LIN {X 0,Y 303.808,Z 469.093,A -85,B 0,C 180,E1 -15922.691,E2 -15922.691} C_VEL
LIN {X 0,Y 303.618,Z 471.715,A -85,B 0,C 180,E1 -15924.688,E2 -15924.688} C_VEL
LIN {X 0,Y 303.612,Z 472.958,A -85,B 0,C 180,E1 -15926.018,E2 -15926.018} C_VEL
LIN {X 0,Y 303.631,Z 473.753,A -85,B 0,C 180,E1 -15927.347,E2 -15927.347} C_VEL
LIN {X 0,Y 303.609,Z 474.149,A -85,B 0,C 180,E1 -15928.674,E2 -15928.674} C_VEL
LIN {X 0,Y 303.653,Z 474.153,A -85,B 0,C 180,E1 -15930,E2 -15930} C_VEL
LIN {X 0,Y 303.62,Z 473.754,A -85,B 0,C 180,E1 -15931.326,E2 -15931.326} C_VEL
LIN {X 0,Y 303.636,Z 472.908,A -85,B 0,C 180,E1 -15932.653,E2 -15932.653} C_VEL
LIN {X 0,Y 303.645,Z 471.649,A -85,B 0,C 180,E1 -15933.982,E2 -15933.982} C_VEL
LIN {X 0,Y 303.681,Z 469.543,A -85,B 0,C 180,E1 -15935.611,E2 -15935.611} C_VEL
LIN {X 0,Y 303.944,Z 465.201,A -85,B 0,C 180,E1 -15937.975,E2 -15937.975} C_VEL
LIN {X 0,Y 304.361,Z 460.303,A -85,B 0,C 180,E1 -15939.973,E2 -15939.973} C_VEL
LIN {X 0,Y 304.994,Z 454.106,A -85,B 0,C 180,E1 -15941.969,E2 -15941.969} C_VEL
LIN {X 0,Y 306.125,Z 446.4,A -85,B 0,C 180,E1 -15943.949,E2 -15943.949} C_VEL
LIN {X 0,Y 307.197,Z 438.485,A -85,B 0,C 180,E1 -15945.593,E2 -15945.593} C_VEL
LIN {X 0,Y 308.389,Z 428.8,A -85,B 0,C 180,E1 -15947.233,E2 -15947.233} C_VEL
LIN {X 0,Y 309.728,Z 418.066,A -85,B 0,C 180,E1 -15948.693,E2 -15948.693} C_VEL
LIN {X 0,Y 310.965,Z 407.709,A -85,B 0,C 180,E1 -15949.816,E2 -15949.816} C_VEL
LIN {X 0,Y 312.28,Z 395.367,A -85,B 0,C 180,E1 -15950.846,E2 -15950.846} C_VEL
LIN {X 0,Y 313.335,Z 382.457,A -85,B 0,C 180,E1 -15951.634,E2 -15951.634} C_VEL
LIN {X 0,Y 314.078,Z 370.101,A -85,B 0,C 180,E1 -15952.142,E2 -15952.142} C_VEL
LIN {X 0,Y 315.753,Z 303.823,A -85,B 0,C 180,E1 -15953.743,E2 -15953.743} C_VEL
LIN {X 0,Y 309.938,Z 264.176,A -85,B 0,C 180,E1 -15955.182,E2 -15955.182} C_VEL
LIN {X 0,Y 309.571,Z 261.875,A -85,B 0,C 180,E1 -15955.29,E2 -15955.29} C_VEL
LIN {X 0,Y 309.852,Z 258.307,A -85,B 0,C 180,E1 -15956.25,E2 -15956.25} C_VEL
LIN {X 0,Y 307.948,Z 247.956,A -85,B 0,C 180,E1 -15959.276,E2 -15959.276} C_VEL
LIN {X 0,Y 305.49,Z 236.432,A -85,B 0,C 180,E1 -15962.824,E2 -15962.824} C_VEL
LIN {X 0,Y 305.461,Z 236.433,A -85,B 0,C 180,E1 -15966.74,E2 -15966.74} C_VEL
LIN {X 0,Y 305.404,Z 236.442,A -85,B 0,C 180,E1 -15970.581,E2 -15970.581} C_VEL
LIN {X 0,Y 305.395,Z 236.443,A -85,B 0,C 180,E1 -15974.481,E2 -15974.481} C_VEL
LIN {X 0,Y 305.398,Z 236.443,A -85,B 0,C 180,E1 -15978.129,E2 -15978.129} C_VEL
LIN {X 0,Y 305.438,Z 236.44,A -85,B 0,C 180,E1 -15981.585,E2 -15981.585} C_VEL
LIN {X 0,Y 305.469,Z 236.432,A -85,B 0,C 180,E1 -15984.881,E2 -15984.881} C_VEL
LIN {X 0,Y 305.446,Z 236.435,A -85,B 0,C 180,E1 -15988.355,E2 -15988.355} C_VEL
LIN {X 0,Y 305.456,Z 236.435,A -85,B 0,C 180,E1 -15991.101,E2 -15991.101} C_VEL
LIN {X 0,Y 305.484,Z 236.431,A -85,B 0,C 180,E1 -15994.073,E2 -15994.073} C_VEL
LIN {X 0,Y 305.462,Z 236.431,A -85,B 0,C 180,E1 -15998.393,E2 -15998.393} C_VEL
LIN {X 0,Y 305.521,Z 236.418,A -85,B 0,C 180,E1 -16002.593,E2 -16002.593} C_VEL
LIN {X 0,Y 305.626,Z 236.412,A -85,B 0,C 180,E1 -16005.341,E2 -16005.341} C_VEL
LIN {X 0,Y 305.618,Z 236.417,A -85,B 0,C 180,E1 -16009.392,E2 -16009.392} C_VEL
LIN {X 0,Y 305.734,Z 236.397,A -85,B 0,C 180,E1 -16012.065,E2 -16012.065} C_VEL
LIN {X 0,Y 305.646,Z 236.404,A -85,B 0,C 180,E1 -16014.716,E2 -16014.716} C_VEL
LIN {X 0,Y 305.933,Z 236.367,A -85,B 0,C 180,E1 -16018.676,E2 -16018.676} C_VEL
LIN {X 0,Y 305.925,Z 236.375,A -85,B 0,C 180,E1 -16021.309,E2 -16021.309} C_VEL
LIN {X 0,Y 305.645,Z 236.413,A -85,B 0,C 180,E1 -16025.269,E2 -16025.269} C_VEL
LIN {X 0,Y 305.73,Z 236.399,A -85,B 0,C 180,E1 -16027.92,E2 -16027.92} C_VEL
LIN {X 0,Y 305.579,Z 236.419,A -85,B 0,C 180,E1 -16031.938,E2 -16031.938} C_VEL
LIN {X 0,Y 305.59,Z 236.418,A -85,B 0,C 180,E1 -16035.006,E2 -16035.006} C_VEL
LIN {X 0,Y 305.539,Z 236.425,A -85,B 0,C 180,E1 -16039.428,E2 -16039.428} C_VEL
LIN {X 0,Y 305.462,Z 236.434,A -85,B 0,C 180,E1 -16043.032,E2 -16043.032} C_VEL
LIN {X 0,Y 305.473,Z 236.429,A -85,B 0,C 180,E1 -16046.201,E2 -16046.201} C_VEL
LIN {X 0,Y 305.446,Z 236.432,A -85,B 0,C 180,E1 -16049.035,E2 -16049.035} C_VEL
LIN {X 0,Y 305.431,Z 236.435,A -85,B 0,C 180,E1 -16053.51,E2 -16053.51} C_VEL
LIN {X 0,Y 305.42,Z 236.437,A -85,B 0,C 180,E1 -16056.735,E2 -16056.735} C_VEL
LIN {X 0,Y 305.416,Z 236.439,A -85,B 0,C 180,E1 -16060.593,E2 -16060.593} C_VEL
LIN {X 0,Y 305.376,Z 236.442,A -85,B 0,C 180,E1 -16064.486,E2 -16064.486} C_VEL
LIN {X 0,Y 305.397,Z 236.44,A -85,B 0,C 180,E1 -16068.137,E2 -16068.137} C_VEL
LIN {X 0,Y 305.429,Z 236.439,A -85,B 0,C 180,E1 -16071.592,E2 -16071.592} C_VEL
LIN {X 0,Y 305.413,Z 236.441,A -85,B 0,C 180,E1 -16074.881,E2 -16074.881} C_VEL
LIN {X 0,Y 305.401,Z 236.44,A -85,B 0,C 180,E1 -16078.351,E2 -16078.351} C_VEL
LIN {X 0,Y 305.469,Z 236.437,A -85,B 0,C 180,E1 -16081.109,E2 -16081.109} C_VEL
LIN {X 0,Y 305.521,Z 236.426,A -85,B 0,C 180,E1 -16084.084,E2 -16084.084} C_VEL
LIN {X 0,Y 305.494,Z 236.429,A -85,B 0,C 180,E1 -16088.403,E2 -16088.403} C_VEL
LIN {X 0,Y 305.538,Z 236.428,A -85,B 0,C 180,E1 -16091.215,E2 -16091.215} C_VEL
LIN {X 0,Y 305.592,Z 236.419,A -85,B 0,C 180,E1 -16095.347,E2 -16095.347} C_VEL
LIN {X 0,Y 305.583,Z 236.42,A -85,B 0,C 180,E1 -16099.398,E2 -16099.398} C_VEL
LIN {X 0,Y 305.758,Z 236.395,A -85,B 0,C 180,E1 -16102.073,E2 -16102.073} C_VEL
LIN {X 0,Y 305.639,Z 236.413,A -85,B 0,C 180,E1 -16104.723,E2 -16104.723} C_VEL
LIN {X 0,Y 305.905,Z 236.38,A -85,B 0,C 180,E1 -16108.683,E2 -16108.683} C_VEL
LIN {X 0,Y 305.905,Z 236.38,A -85,B 0,C 180,E1 -16111.316,E2 -16111.316} C_VEL
LIN {X 0,Y 305.767,Z 236.478,A -85,B 0,C 180,E1 -16116.143,E2 -16116.143} C_VEL
LIN {X 0,Y 306.706,Z 241.054,A -85,B 0,C 180,E1 -16117.592,E2 -16117.592} C_VEL
LIN {X 0,Y 315.156,Z 264.98,A -85,B 0,C 180,E1 -16118.847,E2 -16118.847} C_VEL
LIN {X 0,Y 316.427,Z 271.959,A -85,B 0,C 180,E1 -16119.115,E2 -16119.115} C_VEL
LIN {X 0,Y 314.322,Z 348.83,A -85,B 0,C 180,E1 -16120.97,E2 -16120.97} C_VEL
LIN {X 0,Y 313.559,Z 362.432,A -85,B 0,C 180,E1 -16121.565,E2 -16121.565} C_VEL
LIN {X 0,Y 312.712,Z 375.269,A -85,B 0,C 180,E1 -16122.41,E2 -16122.41} C_VEL
LIN {X 0,Y 311.564,Z 387.718,A -85,B 0,C 180,E1 -16123.523,E2 -16123.523} C_VEL
LIN {X 0,Y 310.355,Z 398.515,A -85,B 0,C 180,E1 -16124.759,E2 -16124.759} C_VEL
LIN {X 0,Y 309.13,Z 408.276,A -85,B 0,C 180,E1 -16126.148,E2 -16126.148} C_VEL
LIN {X 0,Y 307.919,Z 416.664,A -85,B 0,C 180,E1 -16127.602,E2 -16127.602} C_VEL
LIN {X 0,Y 306.806,Z 425.084,A -85,B 0,C 180,E1 -16129.399,E2 -16129.399} C_VEL
LIN {X 0,Y 305.666,Z 433.288,A -85,B 0,C 180,E1 -16131.584,E2 -16131.584} C_VEL
LIN {X 0,Y 304.82,Z 439.711,A -85,B 0,C 180,E1 -16133.795,E2 -16133.795} C_VEL
LIN {X 0,Y 304.268,Z 444.645,A -85,B 0,C 180,E1 -16136.03,E2 -16136.03} C_VEL
LIN {X 0,Y 304.04,Z 447.221,A -85,B 0,C 180,E1 -16137.535,E2 -16137.535} C_VEL
LIN {X 0,Y 303.695,Z 449.214,A -85,B 0,C 180,E1 -16139.075,E2 -16139.075} C_VEL
LIN {X 0,Y 303.446,Z 450.963,A -85,B 0,C 180,E1 -16141.045,E2 -16141.045} C_VEL
LIN {X 0,Y 303.388,Z 451.891,A -85,B 0,C 180,E1 -16143.513,E2 -16143.513} C_VEL
LIN {X 0,Y 303.557,Z 451.493,A -85,B 0,C 180,E1 -16145.89,E2 -16145.89} C_VEL
LIN {X 0,Y 303.919,Z 449.867,A -85,B 0,C 180,E1 -16148.181,E2 -16148.181} C_VEL
LIN {X 0,Y 304.479,Z 447.101,A -85,B 0,C 180,E1 -16150.401,E2 -16150.401} C_VEL
LIN {X 0,Y 305.174,Z 443.252,A -85,B 0,C 180,E1 -16152.543,E2 -16152.543} C_VEL
LIN {X 0,Y 306.16,Z 438.196,A -85,B 0,C 180,E1 -16154.648,E2 -16154.648} C_VEL
LIN {X 0,Y 307.427,Z 431.82,A -85,B 0,C 180,E1 -16156.713,E2 -16156.713} C_VEL
LIN {X 0,Y 308.973,Z 423.866,A -85,B 0,C 180,E1 -16158.74,E2 -16158.74} C_VEL
LIN {X 0,Y 310.631,Z 414.677,A -85,B 0,C 180,E1 -16160.599,E2 -16160.599} C_VEL
LIN {X 0,Y 312.313,Z 405.038,A -85,B 0,C 180,E1 -16162.166,E2 -16162.166} C_VEL
LIN {X 0,Y 313.851,Z 394.716,A -85,B 0,C 180,E1 -16163.516,E2 -16163.516} C_VEL
LIN {X 0,Y 315.441,Z 382.749,A -85,B 0,C 180,E1 -16164.74,E2 -16164.74} C_VEL
LIN {X 0,Y 316.716,Z 370.283,A -85,B 0,C 180,E1 -16165.717,E2 -16165.717} C_VEL
LIN {X 0,Y 317.728,Z 357.146,A -85,B 0,C 180,E1 -16166.439,E2 -16166.439} C_VEL
LIN {X 0,Y 318.347,Z 344.513,A -85,B 0,C 180,E1 -16166.887,E2 -16166.887} C_VEL
LIN {X 0,Y 318.017,Z 338.724,A -85,B 0,C 180,E1 -16167.093,E2 -16167.093} C_VEL
LIN {X 0,Y 313.501,Z 320.095,A -85,B 0,C 180,E1 -16168.037,E2 -16168.037} C_VEL
LIN {X 0,Y 313.101,Z 314.293,A -85,B 0,C 180,E1 -16168.235,E2 -16168.235} C_VEL
LIN {X 0,Y 314.444,Z 274.419,A -85,B 0,C 180,E1 -16169.216,E2 -16169.216} C_VEL
LIN {X 0,Y 309.017,Z 261.151,A -85,B 0,C 180,E1 -16170.202,E2 -16170.202} C_VEL
LIN {X 0,Y 302.527,Z 247.643,A -85,B 0,C 180,E1 -16171.381,E2 -16171.381} C_VEL
LIN {X 0,Y 299.66,Z 242.008,A -85,B 0,C 180,E1 -16171.942,E2 -16171.942} C_VEL
LIN {X 0,Y 298.473,Z 237.305,A -85,B 0,C 180,E1 -16173.695,E2 -16173.695} C_VEL
LIN {X 0,Y 298.405,Z 237.314,A -85,B 0,C 180,E1 -16177.872,E2 -16177.872} C_VEL
LIN {X 0,Y 298.516,Z 237.302,A -85,B 0,C 180,E1 -16180.765,E2 -16180.765} C_VEL
LIN {X 0,Y 298.574,Z 237.292,A -85,B 0,C 180,E1 -16185.003,E2 -16185.003} C_VEL
LIN {X 0,Y 298.576,Z 237.292,A -85,B 0,C 180,E1 -16189.154,E2 -16189.154} C_VEL
LIN {X 0,Y 298.702,Z 237.272,A -85,B 0,C 180,E1 -16191.893,E2 -16191.893} C_VEL
LIN {X 0,Y 298.633,Z 237.281,A -85,B 0,C 180,E1 -16194.606,E2 -16194.606} C_VEL
LIN {X 0,Y 298.91,Z 237.245,A -85,B 0,C 180,E1 -16198.66,E2 -16198.66} C_VEL
LIN {X 0,Y 298.907,Z 237.245,A -85,B 0,C 180,E1 -16201.355,E2 -16201.355} C_VEL
LIN {X 0,Y 298.748,Z 237.264,A -85,B 0,C 180,E1 -16206.762,E2 -16206.762} C_VEL
LIN {X 0,Y 298.623,Z 237.279,A -85,B 0,C 180,E1 -16209.489,E2 -16209.489} C_VEL
LIN {X 0,Y 298.543,Z 237.291,A -85,B 0,C 180,E1 -16213.623,E2 -16213.623} C_VEL
LIN {X 0,Y 298.485,Z 237.306,A -85,B 0,C 180,E1 -16216.419,E2 -16216.419} C_VEL
LIN {X 0,Y 298.443,Z 237.306,A -85,B 0,C 180,E1 -16219.622,E2 -16219.622} C_VEL
LIN {X 0,Y 298.389,Z 237.312,A -85,B 0,C 180,E1 -16223.61,E2 -16223.61} C_VEL
LIN {X 0,Y 298.407,Z 237.306,A -85,B 0,C 180,E1 -16226.589,E2 -16226.589} C_VEL
LIN {X 0,Y 298.363,Z 237.313,A -85,B 0,C 180,E1 -16229.654,E2 -16229.654} C_VEL
LIN {X 0,Y 298.4,Z 237.31,A -85,B 0,C 180,E1 -16232.806,E2 -16232.806} C_VEL
LIN {X 0,Y 298.412,Z 237.312,A -85,B 0,C 180,E1 -16236.078,E2 -16236.078} C_VEL
LIN {X 0,Y 298.355,Z 237.317,A -85,B 0,C 180,E1 -16239.502,E2 -16239.502} C_VEL
LIN {X 0,Y 298.353,Z 237.324,A -85,B 0,C 180,E1 -16243.096,E2 -16243.096} C_VEL
LIN {X 0,Y 298.354,Z 237.323,A -85,B 0,C 180,E1 -16246.913,E2 -16246.913} C_VEL
LIN {X 0,Y 298.376,Z 237.318,A -85,B 0,C 180,E1 -16251.021,E2 -16251.021} C_VEL
LIN {X 0,Y 298.522,Z 237.477,A -85,B 0,C 180,E1 -16254.14,E2 -16254.14} C_VEL
LIN {X 0,Y 301.257,Z 248.367,A -85,B 0,C 180,E1 -16257.946,E2 -16257.946} C_VEL
LIN {X 0,Y 303.213,Z 257.381,A -85,B 0,C 180,E1 -16260.874,E2 -16260.874} C_VEL
LIN {X 0,Y 303.756,Z 260.098,A -85,B 0,C 180,E1 -16261.647,E2 -16261.647} C_VEL
LIN {X 0,Y 307.237,Z 268.773,A -85,B 0,C 180,E1 -16262.317,E2 -16262.317} C_VEL
LIN {X 0,Y 311.274,Z 289.894,A -85,B 0,C 180,E1 -16263.383,E2 -16263.383} C_VEL
LIN {X 0,Y 313.497,Z 306.34,A -85,B 0,C 180,E1 -16264.084,E2 -16264.084} C_VEL
LIN {X 0,Y 311.413,Z 369.696,A -85,B 0,C 180,E1 -16265.674,E2 -16265.674} C_VEL
LIN {X 0,Y 310.328,Z 383.207,A -85,B 0,C 180,E1 -16266.254,E2 -16266.254} C_VEL
LIN {X 0,Y 308.956,Z 395.991,A -85,B 0,C 180,E1 -16267.074,E2 -16267.074} C_VEL
LIN {X 0,Y 307.42,Z 406.931,A -85,B 0,C 180,E1 -16268.016,E2 -16268.016} C_VEL
LIN {X 0,Y 305.646,Z 418.42,A -85,B 0,C 180,E1 -16269.297,E2 -16269.297} C_VEL
LIN {X 0,Y 303.855,Z 428.82,A -85,B 0,C 180,E1 -16270.756,E2 -16270.756} C_VEL
LIN {X 0,Y 302.135,Z 438.215,A -85,B 0,C 180,E1 -16272.399,E2 -16272.399} C_VEL
LIN {X 0,Y 300.481,Z 447.324,A -85,B 0,C 180,E1 -16274.397,E2 -16274.397} C_VEL
LIN {X 0,Y 299.002,Z 454.708,A -85,B 0,C 180,E1 -16276.406,E2 -16276.406} C_VEL
LIN {X 0,Y 297.913,Z 460.651,A -85,B 0,C 180,E1 -16278.433,E2 -16278.433} C_VEL
LIN {X 0,Y 297.22,Z 465.351,A -85,B 0,C 180,E1 -16280.473,E2 -16280.473} C_VEL
LIN {X 0,Y 296.738,Z 468.945,A -85,B 0,C 180,E1 -16282.515,E2 -16282.515} C_VEL
LIN {X 0,Y 296.533,Z 471.531,A -85,B 0,C 180,E1 -16284.56,E2 -16284.56} C_VEL
LIN {X 0,Y 296.511,Z 472.744,A -85,B 0,C 180,E1 -16285.923,E2 -16285.923} C_VEL
LIN {X 0,Y 296.555,Z 473.516,A -85,B 0,C 180,E1 -16287.283,E2 -16287.283} C_VEL
LIN {X 0,Y 296.527,Z 473.893,A -85,B 0,C 180,E1 -16288.642,E2 -16288.642} C_VEL
LIN {X 0,Y 296.567,Z 473.88,A -85,B 0,C 180,E1 -16290,E2 -16290} C_VEL
LIN {X 0,Y 296.538,Z 473.454,A -85,B 0,C 180,E1 -16291.358,E2 -16291.358} C_VEL
LIN {X 0,Y 296.562,Z 472.584,A -85,B 0,C 180,E1 -16292.717,E2 -16292.717} C_VEL
LIN {X 0,Y 296.544,Z 471.305,A -85,B 0,C 180,E1 -16294.077,E2 -16294.077} C_VEL
LIN {X 0,Y 296.609,Z 469.4,A -85,B 0,C 180,E1 -16295.592,E2 -16295.592} C_VEL
LIN {X 0,Y 296.795,Z 466.181,A -85,B 0,C 180,E1 -16297.483,E2 -16297.483} C_VEL
LIN {X 0,Y 297.152,Z 461.638,A -85,B 0,C 180,E1 -16299.53,E2 -16299.53} C_VEL
LIN {X 0,Y 297.736,Z 455.847,A -85,B 0,C 180,E1 -16301.574,E2 -16301.574} C_VEL
LIN {X 0,Y 298.792,Z 448.573,A -85,B 0,C 180,E1 -16303.604,E2 -16303.604} C_VEL
LIN {X 0,Y 300.074,Z 439.516,A -85,B 0,C 180,E1 -16305.625,E2 -16305.625} C_VEL
LIN {X 0,Y 301.234,Z 430.332,A -85,B 0,C 180,E1 -16307.278,E2 -16307.278} C_VEL
LIN {X 0,Y 302.669,Z 419.78,A -85,B 0,C 180,E1 -16308.794,E2 -16308.794} C_VEL
LIN {X 0,Y 304.075,Z 408.261,A -85,B 0,C 180,E1 -16310.108,E2 -16310.108} C_VEL
LIN {X 0,Y 305.407,Z 396.25,A -85,B 0,C 180,E1 -16311.161,E2 -16311.161} C_VEL
LIN {X 0,Y 306.541,Z 382.972,A -85,B 0,C 180,E1 -16312.006,E2 -16312.006} C_VEL
LIN {X 0,Y 307.353,Z 369.883,A -85,B 0,C 180,E1 -16312.564,E2 -16312.564} C_VEL
LIN {X 0,Y 309.013,Z 304.065,A -85,B 0,C 180,E1 -16314.194,E2 -16314.194} C_VEL
LIN {X 0,Y 302.799,Z 261.719,A -85,B 0,C 180,E1 -16315.784,E2 -16315.784} C_VEL
LIN {X 0,Y 302.622,Z 257.699,A -85,B 0,C 180,E1 -16316.927,E2 -16316.927} C_VEL
LIN {X 0,Y 300.354,Z 246.078,A -85,B 0,C 180,E1 -16320.447,E2 -16320.447} C_VEL
LIN {X 0,Y 298.446,Z 237.311,A -85,B 0,C 180,E1 -16323.296,E2 -16323.296} C_VEL
LIN {X 0,Y 298.436,Z 237.308,A -85,B 0,C 180,E1 -16326.797,E2 -16326.797} C_VEL
LIN {X 0,Y 298.345,Z 237.322,A -85,B 0,C 180,E1 -16331.071,E2 -16331.071} C_VEL
LIN {X 0,Y 298.339,Z 237.322,A -85,B 0,C 180,E1 -16335.025,E2 -16335.025} C_VEL
LIN {X 0,Y 298.346,Z 237.319,A -85,B 0,C 180,E1 -16338.92,E2 -16338.92} C_VEL
LIN {X 0,Y 298.434,Z 237.31,A -85,B 0,C 180,E1 -16343.194,E2 -16343.194} C_VEL
LIN {X 0,Y 298.417,Z 237.315,A -85,B 0,C 180,E1 -16345.575,E2 -16345.575} C_VEL
LIN {X 0,Y 298.375,Z 237.315,A -85,B 0,C 180,E1 -16348.782,E2 -16348.782} C_VEL
LIN {X 0,Y 298.4,Z 237.315,A -85,B 0,C 180,E1 -16351.891,E2 -16351.891} C_VEL
LIN {X 0,Y 298.427,Z 237.309,A -85,B 0,C 180,E1 -16354.912,E2 -16354.912} C_VEL
LIN {X 0,Y 298.396,Z 237.314,A -85,B 0,C 180,E1 -16357.855,E2 -16357.855} C_VEL
LIN {X 0,Y 298.456,Z 237.3,A -85,B 0,C 180,E1 -16360.744,E2 -16360.744} C_VEL
LIN {X 0,Y 298.588,Z 237.286,A -85,B 0,C 180,E1 -16364.988,E2 -16364.988} C_VEL
LIN {X 0,Y 298.578,Z 237.292,A -85,B 0,C 180,E1 -16369.139,E2 -16369.139} C_VEL
LIN {X 0,Y 298.68,Z 237.277,A -85,B 0,C 180,E1 -16371.877,E2 -16371.877} C_VEL
LIN {X 0,Y 298.617,Z 237.278,A -85,B 0,C 180,E1 -16374.591,E2 -16374.591} C_VEL
LIN {X 0,Y 298.899,Z 237.242,A -85,B 0,C 180,E1 -16378.645,E2 -16378.645} C_VEL
LIN {X 0,Y 298.893,Z 237.251,A -85,B 0,C 180,E1 -16381.34,E2 -16381.34} C_VEL
LIN {X 0,Y 298.718,Z 237.273,A -85,B 0,C 180,E1 -16386.748,E2 -16386.748} C_VEL
LIN {X 0,Y 298.61,Z 237.287,A -85,B 0,C 180,E1 -16389.474,E2 -16389.474} C_VEL
LIN {X 0,Y 298.525,Z 237.3,A -85,B 0,C 180,E1 -16393.608,E2 -16393.608} C_VEL
LIN {X 0,Y 298.466,Z 237.303,A -85,B 0,C 180,E1 -16396.404,E2 -16396.404} C_VEL
LIN {X 0,Y 298.476,Z 237.304,A -85,B 0,C 180,E1 -16399.639,E2 -16399.639} C_VEL
LIN {X 0,Y 298.4,Z 237.315,A -85,B 0,C 180,E1 -16403.593,E2 -16403.593} C_VEL
LIN {X 0,Y 298.427,Z 237.306,A -85,B 0,C 180,E1 -16406.57,E2 -16406.57} C_VEL
LIN {X 0,Y 298.377,Z 237.307,A -85,B 0,C 180,E1 -16409.635,E2 -16409.635} C_VEL
LIN {X 0,Y 298.36,Z 237.307,A -85,B 0,C 180,E1 -16412.793,E2 -16412.793} C_VEL
LIN {X 0,Y 298.394,Z 237.312,A -85,B 0,C 180,E1 -16416.796,E2 -16416.796} C_VEL
LIN {X 0,Y 298.349,Z 237.322,A -85,B 0,C 180,E1 -16421.081,E2 -16421.081} C_VEL
LIN {X 0,Y 298.359,Z 237.32,A -85,B 0,C 180,E1 -16423.097,E2 -16423.097} C_VEL
LIN {X 0,Y 298.361,Z 237.319,A -85,B 0,C 180,E1 -16426.915,E2 -16426.915} C_VEL
LIN {X 0,Y 298.358,Z 237.318,A -85,B 0,C 180,E1 -16431.001,E2 -16431.001} C_VEL
LIN {X 0,Y 298.37,Z 237.317,A -85,B 0,C 180,E1 -16433.924,E2 -16433.924} C_VEL
LIN {X 0,Y 298.345,Z 237.32,A -85,B 0,C 180,E1 -16437.979,E2 -16437.979} C_VEL
LIN {X 0,Y 298.418,Z 237.31,A -85,B 0,C 180,E1 -16441.9,E2 -16441.9} C_VEL
LIN {X 0,Y 298.447,Z 237.311,A -85,B 0,C 180,E1 -16444.921,E2 -16444.921} C_VEL
LIN {X 0,Y 298.423,Z 237.31,A -85,B 0,C 180,E1 -16447.864,E2 -16447.864} C_VEL
LIN {X 0,Y 298.504,Z 237.303,A -85,B 0,C 180,E1 -16450.755,E2 -16450.755} C_VEL
LIN {X 0,Y 298.537,Z 237.301,A -85,B 0,C 180,E1 -16454.992,E2 -16454.992} C_VEL
LIN {X 0,Y 298.538,Z 237.299,A -85,B 0,C 180,E1 -16459.145,E2 -16459.145} C_VEL
LIN {X 0,Y 298.703,Z 237.274,A -85,B 0,C 180,E1 -16461.885,E2 -16461.885} C_VEL
LIN {X 0,Y 298.609,Z 237.288,A -85,B 0,C 180,E1 -16464.598,E2 -16464.598} C_VEL
LIN {X 0,Y 298.871,Z 237.256,A -85,B 0,C 180,E1 -16468.653,E2 -16468.653} C_VEL
LIN {X 0,Y 298.871,Z 237.256,A -85,B 0,C 180,E1 -16471.347,E2 -16471.347} C_VEL
LIN {X 0,Y 298.655,Z 237.315,A -85,B 0,C 180,E1 -16475.74,E2 -16475.74} C_VEL
LIN {X 0,Y 299.529,Z 241.265,A -85,B 0,C 180,E1 -16477.034,E2 -16477.034} C_VEL
LIN {X 0,Y 308.776,Z 267.168,A -85,B 0,C 180,E1 -16478.446,E2 -16478.446} C_VEL
LIN {X 0,Y 309.771,Z 273.543,A -85,B 0,C 180,E1 -16478.685,E2 -16478.685} C_VEL
LIN {X 0,Y 307.638,Z 348.571,A -85,B 0,C 180,E1 -16480.53,E2 -16480.53} C_VEL
LIN {X 0,Y 306.868,Z 361.957,A -85,B 0,C 180,E1 -16481.117,E2 -16481.117} C_VEL
LIN {X 0,Y 306.044,Z 374.352,A -85,B 0,C 180,E1 -16481.927,E2 -16481.927} C_VEL
LIN {X 0,Y 304.91,Z 386.352,A -85,B 0,C 180,E1 -16482.987,E2 -16482.987} C_VEL
LIN {X 0,Y 303.643,Z 397.605,A -85,B 0,C 180,E1 -16484.269,E2 -16484.269} C_VEL
LIN {X 0,Y 302.363,Z 407.51,A -85,B 0,C 180,E1 -16485.676,E2 -16485.676} C_VEL
LIN {X 0,Y 301.03,Z 416.68,A -85,B 0,C 180,E1 -16487.276,E2 -16487.276} C_VEL
LIN {X 0,Y 299.839,Z 425.328,A -85,B 0,C 180,E1 -16489.156,E2 -16489.156} C_VEL
LIN {X 0,Y 298.667,Z 433.533,A -85,B 0,C 180,E1 -16491.39,E2 -16491.39} C_VEL
LIN {X 0,Y 297.779,Z 439.964,A -85,B 0,C 180,E1 -16493.654,E2 -16493.654} C_VEL
LIN {X 0,Y 297.168,Z 445.08,A -85,B 0,C 180,E1 -16496.037,E2 -16496.037} C_VEL
LIN {X 0,Y 296.783,Z 448.544,A -85,B 0,C 180,E1 -16498.268,E2 -16498.268} C_VEL
LIN {X 0,Y 296.49,Z 450.281,A -85,B 0,C 180,E1 -16499.853,E2 -16499.853} C_VEL
LIN {X 0,Y 296.318,Z 451.458,A -85,B 0,C 180,E1 -16501.451,E2 -16501.451} C_VEL
LIN {X 0,Y 296.303,Z 452.196,A -85,B 0,C 180,E1 -16503.903,E2 -16503.903} C_VEL
LIN {X 0,Y 296.51,Z 451.605,A -85,B 0,C 180,E1 -16506.338,E2 -16506.338} C_VEL
LIN {X 0,Y 296.924,Z 449.847,A -85,B 0,C 180,E1 -16508.656,E2 -16508.656} C_VEL
LIN {X 0,Y 297.57,Z 446.95,A -85,B 0,C 180,E1 -16510.922,E2 -16510.922} C_VEL
LIN {X 0,Y 298.356,Z 442.965,A -85,B 0,C 180,E1 -16513.109,E2 -16513.109} C_VEL
LIN {X 0,Y 299.401,Z 437.791,A -85,B 0,C 180,E1 -16515.249,E2 -16515.249} C_VEL
LIN {X 0,Y 300.765,Z 431.26,A -85,B 0,C 180,E1 -16517.354,E2 -16517.354} C_VEL
LIN {X 0,Y 302.419,Z 423.097,A -85,B 0,C 180,E1 -16519.419,E2 -16519.419} C_VEL
LIN {X 0,Y 304.049,Z 414.684,A -85,B 0,C 180,E1 -16521.131,E2 -16521.131} C_VEL
LIN {X 0,Y 305.787,Z 405.006,A -85,B 0,C 180,E1 -16522.728,E2 -16522.728} C_VEL
LIN {X 0,Y 307.441,Z 394.349,A -85,B 0,C 180,E1 -16524.13,E2 -16524.13} C_VEL
LIN {X 0,Y 309.116,Z 382.252,A -85,B 0,C 180,E1 -16525.373,E2 -16525.373} C_VEL
LIN {X 0,Y 310.324,Z 371.025,A -85,B 0,C 180,E1 -16526.262,E2 -16526.262} C_VEL
LIN {X 0,Y 311.385,Z 357.871,A -85,B 0,C 180,E1 -16527.01,E2 -16527.01} C_VEL
LIN {X 0,Y 312.073,Z 344.69,A -85,B 0,C 180,E1 -16527.488,E2 -16527.488} C_VEL
LIN {X 0,Y 313.101,Z 314.293,A -85,B 0,C 180,E1 -16528.235,E2 -16528.235} C_VEL
LIN {X 0,Y 312.723,Z 308.495,A -85,B 0,C 180,E1 -16528.438,E2 -16528.438} C_VEL
LIN {X 0,Y 308.404,Z 289.883,A -85,B 0,C 180,E1 -16529.436,E2 -16529.436} C_VEL
LIN {X 0,Y 308.061,Z 284.086,A -85,B 0,C 180,E1 -16529.642,E2 -16529.642} C_VEL
LIN {X 0,Y 308.218,Z 275.788,A -85,B 0,C 180,E1 -16529.866,E2 -16529.866} C_VEL
LIN {X 0,Y 302.127,Z 261.5,A -85,B 0,C 180,E1 -16531.007,E2 -16531.007} C_VEL
LIN {X 0,Y 296.111,Z 249.265,A -85,B 0,C 180,E1 -16532.153,E2 -16532.153} C_VEL
LIN {X 0,Y 292.491,Z 242.304,A -85,B 0,C 180,E1 -16532.904,E2 -16532.904} C_VEL
LIN {X 0,Y 291.428,Z 238.184,A -85,B 0,C 180,E1 -16534.523,E2 -16534.523} C_VEL
LIN {X 0,Y 291.356,Z 238.194,A -85,B 0,C 180,E1 -16537.307,E2 -16537.307} C_VEL
LIN {X 0,Y 291.436,Z 238.182,A -85,B 0,C 180,E1 -16540.278,E2 -16540.278} C_VEL
LIN {X 0,Y 291.522,Z 238.173,A -85,B 0,C 180,E1 -16544.642,E2 -16544.642} C_VEL
LIN {X 0,Y 291.52,Z 238.169,A -85,B 0,C 180,E1 -16548.889,E2 -16548.889} C_VEL
LIN {X 0,Y 291.652,Z 238.15,A -85,B 0,C 180,E1 -16551.695,E2 -16551.695} C_VEL
LIN {X 0,Y 291.602,Z 238.156,A -85,B 0,C 180,E1 -16554.476,E2 -16554.476} C_VEL
LIN {X 0,Y 291.876,Z 238.12,A -85,B 0,C 180,E1 -16558.628,E2 -16558.628} C_VEL
LIN {X 0,Y 291.873,Z 238.121,A -85,B 0,C 180,E1 -16561.387,E2 -16561.387} C_VEL
LIN {X 0,Y 291.699,Z 238.143,A -85,B 0,C 180,E1 -16566.926,E2 -16566.926} C_VEL
LIN {X 0,Y 291.566,Z 238.157,A -85,B 0,C 180,E1 -16569.721,E2 -16569.721} C_VEL
LIN {X 0,Y 291.514,Z 238.164,A -85,B 0,C 180,E1 -16573.958,E2 -16573.958} C_VEL
LIN {X 0,Y 291.43,Z 238.182,A -85,B 0,C 180,E1 -16576.828,E2 -16576.828} C_VEL
LIN {X 0,Y 291.395,Z 238.184,A -85,B 0,C 180,E1 -16579.849,E2 -16579.849} C_VEL
LIN {X 0,Y 291.334,Z 238.193,A -85,B 0,C 180,E1 -16584.218,E2 -16584.218} C_VEL
LIN {X 0,Y 291.335,Z 238.19,A -85,B 0,C 180,E1 -16587.287,E2 -16587.287} C_VEL
LIN {X 0,Y 291.308,Z 238.191,A -85,B 0,C 180,E1 -16590.447,E2 -16590.447} C_VEL
LIN {X 0,Y 291.352,Z 238.185,A -85,B 0,C 180,E1 -16593.704,E2 -16593.704} C_VEL
LIN {X 0,Y 291.358,Z 238.188,A -85,B 0,C 180,E1 -16597.251,E2 -16597.251} C_VEL
LIN {X 0,Y 291.296,Z 238.201,A -85,B 0,C 180,E1 -16600.656,E2 -16600.656} C_VEL
LIN {X 0,Y 291.288,Z 238.204,A -85,B 0,C 180,E1 -16604.41,E2 -16604.41} C_VEL
LIN {X 0,Y 291.286,Z 238.207,A -85,B 0,C 180,E1 -16608.421,E2 -16608.421} C_VEL
LIN {X 0,Y 291.327,Z 238.196,A -85,B 0,C 180,E1 -16611.156,E2 -16611.156} C_VEL
LIN {X 0,Y 291.425,Z 238.309,A -85,B 0,C 180,E1 -16613.301,E2 -16613.301} C_VEL
LIN {X 0,Y 293.758,Z 247.319,A -85,B 0,C 180,E1 -16616.616,E2 -16616.616} C_VEL
LIN {X 0,Y 295.839,Z 256.274,A -85,B 0,C 180,E1 -16619.678,E2 -16619.678} C_VEL
LIN {X 0,Y 296.516,Z 259.545,A -85,B 0,C 180,E1 -16620.724,E2 -16620.724} C_VEL
LIN {X 0,Y 301.443,Z 271.272,A -85,B 0,C 180,E1 -16621.705,E2 -16621.705} C_VEL
LIN {X 0,Y 305.198,Z 291.302,A -85,B 0,C 180,E1 -16622.745,E2 -16622.745} C_VEL
LIN {X 0,Y 307.345,Z 306.594,A -85,B 0,C 180,E1 -16623.433,E2 -16623.433} C_VEL
LIN {X 0,Y 305.173,Z 369.226,A -85,B 0,C 180,E1 -16625.042,E2 -16625.042} C_VEL
LIN {X 0,Y 304.048,Z 382.944,A -85,B 0,C 180,E1 -16625.642,E2 -16625.642} C_VEL
LIN {X 0,Y 302.606,Z 395.724,A -85,B 0,C 180,E1 -16626.474,E2 -16626.474} C_VEL
LIN {X 0,Y 300.879,Z 407.449,A -85,B 0,C 180,E1 -16627.513,E2 -16627.513} C_VEL
LIN {X 0,Y 299.046,Z 418.797,A -85,B 0,C 180,E1 -16628.819,E2 -16628.819} C_VEL
LIN {X 0,Y 297.175,Z 429.085,A -85,B 0,C 180,E1 -16630.306,E2 -16630.306} C_VEL
LIN {X 0,Y 295.345,Z 438.359,A -85,B 0,C 180,E1 -16631.981,E2 -16631.981} C_VEL
LIN {X 0,Y 293.618,Z 447.401,A -85,B 0,C 180,E1 -16634.023,E2 -16634.023} C_VEL
LIN {X 0,Y 292.094,Z 454.715,A -85,B 0,C 180,E1 -16636.078,E2 -16636.078} C_VEL
LIN {X 0,Y 290.925,Z 460.588,A -85,B 0,C 180,E1 -16638.151,E2 -16638.151} C_VEL
LIN {X 0,Y 290.177,Z 465.234,A -85,B 0,C 180,E1 -16640.239,E2 -16640.239} C_VEL
LIN {X 0,Y 289.689,Z 468.794,A -85,B 0,C 180,E1 -16642.332,E2 -16642.332} C_VEL
LIN {X 0,Y 289.452,Z 471.527,A -85,B 0,C 180,E1 -16644.606,E2 -16644.606} C_VEL
LIN {X 0,Y 289.479,Z 473.279,A -85,B 0,C 180,E1 -16647.217,E2 -16647.217} C_VEL
LIN {X 0,Y 289.448,Z 473.639,A -85,B 0,C 180,E1 -16648.609,E2 -16648.609} C_VEL
LIN {X 0,Y 289.483,Z 473.608,A -85,B 0,C 180,E1 -16650,E2 -16650} C_VEL
LIN {X 0,Y 289.458,Z 473.145,A -85,B 0,C 180,E1 -16651.391,E2 -16651.391} C_VEL
LIN {X 0,Y 289.487,Z 472.255,A -85,B 0,C 180,E1 -16652.783,E2 -16652.783} C_VEL
LIN {X 0,Y 289.5,Z 469.344,A -85,B 0,C 180,E1 -16655.493,E2 -16655.493} C_VEL
LIN {X 0,Y 289.724,Z 465.767,A -85,B 0,C 180,E1 -16657.667,E2 -16657.667} C_VEL
LIN {X 0,Y 290.118,Z 461.175,A -85,B 0,C 180,E1 -16659.763,E2 -16659.763} C_VEL
LIN {X 0,Y 290.897,Z 454.181,A -85,B 0,C 180,E1 -16662.204,E2 -16662.204} C_VEL
LIN {X 0,Y 292.061,Z 446.601,A -85,B 0,C 180,E1 -16664.279,E2 -16664.279} C_VEL
LIN {X 0,Y 293.192,Z 438.847,A -85,B 0,C 180,E1 -16666.001,E2 -16666.001} C_VEL
LIN {X 0,Y 294.459,Z 429.385,A -85,B 0,C 180,E1 -16667.716,E2 -16667.716} C_VEL
LIN {X 0,Y 295.866,Z 418.864,A -85,B 0,C 180,E1 -16669.243,E2 -16669.243} C_VEL
LIN {X 0,Y 297.375,Z 407.207,A -85,B 0,C 180,E1 -16670.581,E2 -16670.581} C_VEL
LIN {X 0,Y 298.774,Z 394.868,A -85,B 0,C 180,E1 -16671.654,E2 -16671.654} C_VEL
LIN {X 0,Y 299.894,Z 381.969,A -85,B 0,C 180,E1 -16672.475,E2 -16672.475} C_VEL
LIN {X 0,Y 300.661,Z 369.638,A -85,B 0,C 180,E1 -16673.004,E2 -16673.004} C_VEL
LIN {X 0,Y 302.347,Z 304.812,A -85,B 0,C 180,E1 -16674.648,E2 -16674.648} C_VEL
LIN {X 0,Y 296.876,Z 267.069,A -85,B 0,C 180,E1 -16676.098,E2 -16676.098} C_VEL
LIN {X 0,Y 295.954,Z 261.323,A -85,B 0,C 180,E1 -16676.369,E2 -16676.369} C_VEL
LIN {X 0,Y 294.494,Z 253.019,A -85,B 0,C 180,E1 -16678.898,E2 -16678.898} C_VEL
LIN {X 0,Y 292.524,Z 243.518,A -85,B 0,C 180,E1 -16681.907,E2 -16681.907} C_VEL
LIN {X 0,Y 291.404,Z 238.188,A -85,B 0,C 180,E1 -16683.69,E2 -16683.69} C_VEL
LIN {X 0,Y 291.356,Z 238.191,A -85,B 0,C 180,E1 -16687.24,E2 -16687.24} C_VEL
LIN {X 0,Y 291.296,Z 238.2,A -85,B 0,C 180,E1 -16690.647,E2 -16690.647} C_VEL
LIN {X 0,Y 291.265,Z 238.204,A -85,B 0,C 180,E1 -16694.405,E2 -16694.405} C_VEL
LIN {X 0,Y 291.284,Z 238.2,A -85,B 0,C 180,E1 -16698.412,E2 -16698.412} C_VEL
LIN {X 0,Y 291.324,Z 238.195,A -85,B 0,C 180,E1 -16701.146,E2 -16701.146} C_VEL
LIN {X 0,Y 291.365,Z 238.189,A -85,B 0,C 180,E1 -16704.619,E2 -16704.619} C_VEL
LIN {X 0,Y 291.372,Z 238.19,A -85,B 0,C 180,E1 -16707.944,E2 -16707.944} C_VEL
LIN {X 0,Y 291.32,Z 238.196,A -85,B 0,C 180,E1 -16711.145,E2 -16711.145} C_VEL
LIN {X 0,Y 291.352,Z 238.19,A -85,B 0,C 180,E1 -16714.259,E2 -16714.259} C_VEL
LIN {X 0,Y 291.355,Z 238.192,A -85,B 0,C 180,E1 -16717.29,E2 -16717.29} C_VEL
LIN {X 0,Y 291.389,Z 238.18,A -85,B 0,C 180,E1 -16720.258,E2 -16720.258} C_VEL
LIN {X 0,Y 291.5,Z 238.167,A -85,B 0,C 180,E1 -16724.659,E2 -16724.659} C_VEL
LIN {X 0,Y 291.524,Z 238.169,A -85,B 0,C 180,E1 -16728.873,E2 -16728.873} C_VEL
LIN {X 0,Y 291.627,Z 238.157,A -85,B 0,C 180,E1 -16731.679,E2 -16731.679} C_VEL
LIN {X 0,Y 291.588,Z 238.153,A -85,B 0,C 180,E1 -16734.46,E2 -16734.46} C_VEL
LIN {X 0,Y 291.866,Z 238.117,A -85,B 0,C 180,E1 -16738.612,E2 -16738.612} C_VEL
LIN {X 0,Y 291.861,Z 238.127,A -85,B 0,C 180,E1 -16741.372,E2 -16741.372} C_VEL
LIN {X 0,Y 291.67,Z 238.151,A -85,B 0,C 180,E1 -16746.911,E2 -16746.911} C_VEL
LIN {X 0,Y 291.553,Z 238.165,A -85,B 0,C 180,E1 -16749.706,E2 -16749.706} C_VEL
LIN {X 0,Y 291.496,Z 238.173,A -85,B 0,C 180,E1 -16753.943,E2 -16753.943} C_VEL
LIN {X 0,Y 291.426,Z 238.177,A -85,B 0,C 180,E1 -16758.261,E2 -16758.261} C_VEL
LIN {X 0,Y 291.348,Z 238.192,A -85,B 0,C 180,E1 -16761.203,E2 -16761.203} C_VEL
LIN {X 0,Y 291.346,Z 238.19,A -85,B 0,C 180,E1 -16764.2,E2 -16764.2} C_VEL
LIN {X 0,Y 291.371,Z 238.188,A -85,B 0,C 180,E1 -16767.266,E2 -16767.266} C_VEL
LIN {X 0,Y 291.296,Z 238.185,A -85,B 0,C 180,E1 -16770.431,E2 -16770.431} C_VEL
LIN {X 0,Y 291.31,Z 238.191,A -85,B 0,C 180,E1 -16773.691,E2 -16773.691} C_VEL
LIN {X 0,Y 291.326,Z 238.195,A -85,B 0,C 180,E1 -16777.243,E2 -16777.243} C_VEL
LIN {X 0,Y 291.294,Z 238.198,A -85,B 0,C 180,E1 -16780.636,E2 -16780.636} C_VEL
LIN {X 0,Y 291.254,Z 238.201,A -85,B 0,C 180,E1 -16784.395,E2 -16784.395} C_VEL
LIN {X 0,Y 291.283,Z 238.199,A -85,B 0,C 180,E1 -16788.398,E2 -16788.398} C_VEL
LIN {X 0,Y 291.307,Z 238.198,A -85,B 0,C 180,E1 -16791.152,E2 -16791.152} C_VEL
LIN {X 0,Y 291.314,Z 238.196,A -85,B 0,C 180,E1 -16794.62,E2 -16794.62} C_VEL
LIN {X 0,Y 291.322,Z 238.195,A -85,B 0,C 180,E1 -16797.945,E2 -16797.945} C_VEL
LIN {X 0,Y 291.335,Z 238.198,A -85,B 0,C 180,E1 -16801.154,E2 -16801.154} C_VEL
LIN {X 0,Y 291.376,Z 238.189,A -85,B 0,C 180,E1 -16804.269,E2 -16804.269} C_VEL
LIN {X 0,Y 291.38,Z 238.191,A -85,B 0,C 180,E1 -16807.3,E2 -16807.3} C_VEL
LIN {X 0,Y 291.451,Z 238.18,A -85,B 0,C 180,E1 -16810.27,E2 -16810.27} C_VEL
LIN {X 0,Y 291.486,Z 238.177,A -85,B 0,C 180,E1 -16814.632,E2 -16814.632} C_VEL
LIN {X 0,Y 291.481,Z 238.178,A -85,B 0,C 180,E1 -16818.879,E2 -16818.879} C_VEL
LIN {X 0,Y 291.654,Z 238.153,A -85,B 0,C 180,E1 -16821.687,E2 -16821.687} C_VEL
LIN {X 0,Y 291.579,Z 238.163,A -85,B 0,C 180,E1 -16824.467,E2 -16824.467} C_VEL
LIN {X 0,Y 291.838,Z 238.132,A -85,B 0,C 180,E1 -16828.62,E2 -16828.62} C_VEL
LIN {X 0,Y 291.838,Z 238.132,A -85,B 0,C 180,E1 -16831.38,E2 -16831.38} C_VEL
LIN {X 0,Y 291.575,Z 238.262,A -85,B 0,C 180,E1 -16835.359,E2 -16835.359} C_VEL
LIN {X 0,Y 292.326,Z 241.303,A -85,B 0,C 180,E1 -16836.427,E2 -16836.427} C_VEL
LIN {X 0,Y 301.729,Z 267.231,A -85,B 0,C 180,E1 -16837.918,E2 -16837.918} C_VEL
LIN {X 0,Y 303.118,Z 272.996,A -85,B 0,C 180,E1 -16838.179,E2 -16838.179} C_VEL
LIN {X 0,Y 300.978,Z 348.514,A -85,B 0,C 180,E1 -16840.079,E2 -16840.079} C_VEL
LIN {X 0,Y 300.166,Z 362.268,A -85,B 0,C 180,E1 -16840.693,E2 -16840.693} C_VEL
LIN {X 0,Y 299.288,Z 374.572,A -85,B 0,C 180,E1 -16841.513,E2 -16841.513} C_VEL
LIN {X 0,Y 298.12,Z 386.576,A -85,B 0,C 180,E1 -16842.595,E2 -16842.595} C_VEL
LIN {X 0,Y 296.806,Z 397.94,A -85,B 0,C 180,E1 -16843.919,E2 -16843.919} C_VEL
LIN {X 0,Y 295.339,Z 408.893,A -85,B 0,C 180,E1 -16845.527,E2 -16845.527} C_VEL
LIN {X 0,Y 293.947,Z 418.086,A -85,B 0,C 180,E1 -16847.219,E2 -16847.219} C_VEL
LIN {X 0,Y 292.657,Z 427.08,A -85,B 0,C 180,E1 -16849.28,E2 -16849.28} C_VEL
LIN {X 0,Y 291.673,Z 433.778,A -85,B 0,C 180,E1 -16851.187,E2 -16851.187} C_VEL
LIN {X 0,Y 290.801,Z 439.822,A -85,B 0,C 180,E1 -16853.338,E2 -16853.338} C_VEL
LIN {X 0,Y 290.108,Z 445.167,A -85,B 0,C 180,E1 -16855.852,E2 -16855.852} C_VEL
LIN {X 0,Y 289.691,Z 448.808,A -85,B 0,C 180,E1 -16858.233,E2 -16858.233} C_VEL
LIN {X 0,Y 289.279,Z 451.225,A -85,B 0,C 180,E1 -16860.676,E2 -16860.676} C_VEL
LIN {X 0,Y 289.178,Z 452.098,A -85,B 0,C 180,E1 -16862.321,E2 -16862.321} C_VEL
LIN {X 0,Y 289.218,Z 452.443,A -85,B 0,C 180,E1 -16864.309,E2 -16864.309} C_VEL
LIN {X 0,Y 289.475,Z 451.72,A -85,B 0,C 180,E1 -16866.774,E2 -16866.774} C_VEL
LIN {X 0,Y 289.976,Z 449.821,A -85,B 0,C 180,E1 -16869.16,E2 -16869.16} C_VEL
LIN {X 0,Y 290.646,Z 446.825,A -85,B 0,C 180,E1 -16871.46,E2 -16871.46} C_VEL
LIN {X 0,Y 291.549,Z 442.708,A -85,B 0,C 180,E1 -16873.698,E2 -16873.698} C_VEL
LIN {X 0,Y 292.761,Z 436.862,A -85,B 0,C 180,E1 -16876.068,E2 -16876.068} C_VEL
LIN {X 0,Y 294.371,Z 429.597,A -85,B 0,C 180,E1 -16878.327,E2 -16878.327} C_VEL
LIN {X 0,Y 296.144,Z 421.542,A -85,B 0,C 180,E1 -16880.307,E2 -16880.307} C_VEL
LIN {X 0,Y 298.059,Z 411.818,A -85,B 0,C 180,E1 -16882.201,E2 -16882.201} C_VEL
LIN {X 0,Y 300.02,Z 401.013,A -85,B 0,C 180,E1 -16883.875,E2 -16883.875} C_VEL
LIN {X 0,Y 301.714,Z 390.202,A -85,B 0,C 180,E1 -16885.193,E2 -16885.193} C_VEL
LIN {X 0,Y 303.259,Z 378.261,A -85,B 0,C 180,E1 -16886.329,E2 -16886.329} C_VEL
LIN {X 0,Y 304.553,Z 365.698,A -85,B 0,C 180,E1 -16887.227,E2 -16887.227} C_VEL
LIN {X 0,Y 305.495,Z 353.058,A -85,B 0,C 180,E1 -16887.845,E2 -16887.845} C_VEL
LIN {X 0,Y 306.221,Z 335.077,A -85,B 0,C 180,E1 -16888.367,E2 -16888.367} C_VEL
LIN {X 0,Y 308.061,Z 284.086,A -85,B 0,C 180,E1 -16889.642,E2 -16889.642} C_VEL
LIN {X 0,Y 307.569,Z 281.027,A -85,B 0,C 180,E1 -16889.787,E2 -16889.787} C_VEL
LIN {X 0,Y 305.512,Z 277.354,A -85,B 0,C 180,E1 -16890.131,E2 -16890.131} C_VEL
LIN {X 0,Y 299.08,Z 269.927,A -85,B 0,C 180,E1 -16891.125,E2 -16891.125} C_VEL
LIN {X 0,Y 297.909,Z 267.661,A -85,B 0,C 180,E1 -16891.343,E2 -16891.343} C_VEL
LIN {X 0,Y 291.396,Z 253.964,A -85,B 0,C 180,E1 -16892.639,E2 -16892.639} C_VEL
LIN {X 0,Y 286.807,Z 245.687,A -85,B 0,C 180,E1 -16893.562,E2 -16893.562} C_VEL
LIN {X 0,Y 285.36,Z 242.752,A -85,B 0,C 180,E1 -16893.892,E2 -16893.892} C_VEL
LIN {X 0,Y 284.354,Z 239.065,A -85,B 0,C 180,E1 -16895.447,E2 -16895.447} C_VEL
LIN {X 0,Y 284.366,Z 239.063,A -85,B 0,C 180,E1 -16899.906,E2 -16899.906} C_VEL
LIN {X 0,Y 284.459,Z 239.054,A -85,B 0,C 180,E1 -16904.478,E2 -16904.478} C_VEL
LIN {X 0,Y 284.472,Z 239.046,A -85,B 0,C 180,E1 -16908.61,E2 -16908.61} C_VEL
LIN {X 0,Y 284.606,Z 239.027,A -85,B 0,C 180,E1 -16911.488,E2 -16911.488} C_VEL
LIN {X 0,Y 284.572,Z 239.032,A -85,B 0,C 180,E1 -16914.339,E2 -16914.339} C_VEL
LIN {X 0,Y 284.843,Z 238.996,A -85,B 0,C 180,E1 -16918.594,E2 -16918.594} C_VEL
LIN {X 0,Y 284.839,Z 238.997,A -85,B 0,C 180,E1 -16921.422,E2 -16921.422} C_VEL
LIN {X 0,Y 284.654,Z 239.022,A -85,B 0,C 180,E1 -16927.099,E2 -16927.099} C_VEL
LIN {X 0,Y 284.512,Z 239.034,A -85,B 0,C 180,E1 -16929.965,E2 -16929.965} C_VEL
LIN {X 0,Y 284.463,Z 239.041,A -85,B 0,C 180,E1 -16934.311,E2 -16934.311} C_VEL
LIN {X 0,Y 284.333,Z 239.058,A -85,B 0,C 180,E1 -16938.751,E2 -16938.751} C_VEL
LIN {X 0,Y 284.314,Z 239.063,A -85,B 0,C 180,E1 -16943.305,E2 -16943.305} C_VEL
LIN {X 0,Y 284.292,Z 239.066,A -85,B 0,C 180,E1 -16947.135,E2 -16947.135} C_VEL
LIN {X 0,Y 284.281,Z 239.066,A -85,B 0,C 180,E1 -16950.089,E2 -16950.089} C_VEL
LIN {X 0,Y 284.295,Z 239.066,A -85,B 0,C 180,E1 -16952.954,E2 -16952.954} C_VEL
LIN {X 0,Y 284.326,Z 239.064,A -85,B 0,C 180,E1 -16956.394,E2 -16956.394} C_VEL
LIN {X 0,Y 284.266,Z 239.072,A -85,B 0,C 180,E1 -16960.009,E2 -16960.009} C_VEL
LIN {X 0,Y 284.236,Z 239.084,A -85,B 0,C 180,E1 -16964.19,E2 -16964.19} C_VEL
LIN {X 0,Y 284.231,Z 239.086,A -85,B 0,C 180,E1 -16968.118,E2 -16968.118} C_VEL
LIN {X 0,Y 284.295,Z 239.072,A -85,B 0,C 180,E1 -16972.294,E2 -16972.294} C_VEL
LIN {X 0,Y 286.128,Z 245.579,A -85,B 0,C 180,E1 -16974.911,E2 -16974.911} C_VEL
LIN {X 0,Y 288.765,Z 256.431,A -85,B 0,C 180,E1 -16978.831,E2 -16978.831} C_VEL
LIN {X 0,Y 289.286,Z 259.133,A -85,B 0,C 180,E1 -16979.733,E2 -16979.733} C_VEL
LIN {X 0,Y 295.669,Z 273.692,A -85,B 0,C 180,E1 -16981.058,E2 -16981.058} C_VEL
LIN {X 0,Y 299.348,Z 293.755,A -85,B 0,C 180,E1 -16982.135,E2 -16982.135} C_VEL
LIN {X 0,Y 301.231,Z 307.511,A -85,B 0,C 180,E1 -16982.769,E2 -16982.769} C_VEL
LIN {X 0,Y 298.996,Z 368.89,A -85,B 0,C 180,E1 -16984.375,E2 -16984.375} C_VEL
LIN {X 0,Y 297.794,Z 382.925,A -85,B 0,C 180,E1 -16985.003,E2 -16985.003} C_VEL
LIN {X 0,Y 296.298,Z 395.586,A -85,B 0,C 180,E1 -16985.849,E2 -16985.849} C_VEL
LIN {X 0,Y 294.369,Z 408.039,A -85,B 0,C 180,E1 -16986.987,E2 -16986.987} C_VEL
LIN {X 0,Y 292.455,Z 419.205,A -85,B 0,C 180,E1 -16988.317,E2 -16988.317} C_VEL
LIN {X 0,Y 290.502,Z 429.324,A -85,B 0,C 180,E1 -16989.834,E2 -16989.834} C_VEL
LIN {X 0,Y 288.583,Z 438.503,A -85,B 0,C 180,E1 -16991.543,E2 -16991.543} C_VEL
LIN {X 0,Y 286.76,Z 447.48,A -85,B 0,C 180,E1 -16993.63,E2 -16993.63} C_VEL
LIN {X 0,Y 285.19,Z 454.73,A -85,B 0,C 180,E1 -16995.734,E2 -16995.734} C_VEL
LIN {X 0,Y 283.952,Z 460.536,A -85,B 0,C 180,E1 -16997.856,E2 -16997.856} C_VEL
LIN {X 0,Y 283.157,Z 465.133,A -85,B 0,C 180,E1 -16999.995,E2 -16999.995} C_VEL
LIN {X 0,Y 282.638,Z 468.649,A -85,B 0,C 180,E1 -17002.14,E2 -17002.14} C_VEL
LIN {X 0,Y 282.376,Z 471.475,A -85,B 0,C 180,E1 -17004.644,E2 -17004.644} C_VEL
LIN {X 0,Y 282.382,Z 473.042,A -85,B 0,C 180,E1 -17007.147,E2 -17007.147} C_VEL
LIN {X 0,Y 282.371,Z 473.385,A -85,B 0,C 180,E1 -17008.574,E2 -17008.574} C_VEL
LIN {X 0,Y 282.401,Z 473.333,A -85,B 0,C 180,E1 -17010,E2 -17010} C_VEL
LIN {X 0,Y 282.38,Z 472.835,A -85,B 0,C 180,E1 -17011.426,E2 -17011.426} C_VEL
LIN {X 0,Y 282.391,Z 471.925,A -85,B 0,C 180,E1 -17012.853,E2 -17012.853} C_VEL
LIN {X 0,Y 282.423,Z 469.195,A -85,B 0,C 180,E1 -17015.457,E2 -17015.457} C_VEL
LIN {X 0,Y 282.66,Z 465.346,A -85,B 0,C 180,E1 -17017.86,E2 -17017.86} C_VEL
LIN {X 0,Y 283.099,Z 460.702,A -85,B 0,C 180,E1 -17020.007,E2 -17020.007} C_VEL
LIN {X 0,Y 283.907,Z 453.641,A -85,B 0,C 180,E1 -17022.509,E2 -17022.509} C_VEL
LIN {X 0,Y 285.104,Z 445.999,A -85,B 0,C 180,E1 -17024.635,E2 -17024.635} C_VEL
LIN {X 0,Y 286.416,Z 437.407,A -85,B 0,C 180,E1 -17026.548,E2 -17026.548} C_VEL
LIN {X 0,Y 287.789,Z 427.501,A -85,B 0,C 180,E1 -17028.325,E2 -17028.325} C_VEL
LIN {X 0,Y 289.323,Z 416.656,A -85,B 0,C 180,E1 -17029.881,E2 -17029.881} C_VEL
LIN {X 0,Y 290.698,Z 406.119,A -85,B 0,C 180,E1 -17031.076,E2 -17031.076} C_VEL
LIN {X 0,Y 292.135,Z 393.481,A -85,B 0,C 180,E1 -17032.172,E2 -17032.172} C_VEL
LIN {X 0,Y 293.31,Z 380.194,A -85,B 0,C 180,E1 -17033.008,E2 -17033.008} C_VEL
LIN {X 0,Y 294.109,Z 366.63,A -85,B 0,C 180,E1 -17033.547,E2 -17033.547} C_VEL
LIN {X 0,Y 295.72,Z 305.593,A -85,B 0,C 180,E1 -17035.12,E2 -17035.12} C_VEL
LIN {X 0,Y 289.956,Z 265.624,A -85,B 0,C 180,E1 -17036.697,E2 -17036.697} C_VEL
LIN {X 0,Y 288.845,Z 261.124,A -85,B 0,C 180,E1 -17036.941,E2 -17036.941} C_VEL
LIN {X 0,Y 286.35,Z 248.268,A -85,B 0,C 180,E1 -17041.024,E2 -17041.024} C_VEL
LIN {X 0,Y 284.341,Z 239.066,A -85,B 0,C 180,E1 -17044.107,E2 -17044.107} C_VEL
LIN {X 0,Y 284.278,Z 239.072,A -85,B 0,C 180,E1 -17048.173,E2 -17048.173} C_VEL
LIN {X 0,Y 284.219,Z 239.082,A -85,B 0,C 180,E1 -17052.105,E2 -17052.105} C_VEL
LIN {X 0,Y 284.221,Z 239.082,A -85,B 0,C 180,E1 -17056.175,E2 -17056.175} C_VEL
LIN {X 0,Y 284.268,Z 239.076,A -85,B 0,C 180,E1 -17060.032,E2 -17060.032} C_VEL
LIN {X 0,Y 284.326,Z 239.07,A -85,B 0,C 180,E1 -17063.606,E2 -17063.606} C_VEL
LIN {X 0,Y 284.296,Z 239.072,A -85,B 0,C 180,E1 -17067.191,E2 -17067.191} C_VEL
LIN {X 0,Y 284.315,Z 239.068,A -85,B 0,C 180,E1 -17070.364,E2 -17070.364} C_VEL
LIN {X 0,Y 284.303,Z 239.071,A -85,B 0,C 180,E1 -17073.572,E2 -17073.572} C_VEL
LIN {X 0,Y 284.315,Z 239.067,A -85,B 0,C 180,E1 -17076.695,E2 -17076.695} C_VEL
LIN {X 0,Y 284.339,Z 239.059,A -85,B 0,C 180,E1 -17079.921,E2 -17079.921} C_VEL
LIN {X 0,Y 284.448,Z 239.045,A -85,B 0,C 180,E1 -17084.487,E2 -17084.487} C_VEL
LIN {X 0,Y 284.462,Z 239.048,A -85,B 0,C 180,E1 -17088.593,E2 -17088.593} C_VEL
LIN {X 0,Y 284.578,Z 239.036,A -85,B 0,C 180,E1 -17091.471,E2 -17091.471} C_VEL
LIN {X 0,Y 284.558,Z 239.027,A -85,B 0,C 180,E1 -17094.323,E2 -17094.323} C_VEL
LIN {X 0,Y 284.832,Z 238.992,A -85,B 0,C 180,E1 -17098.578,E2 -17098.578} C_VEL
LIN {X 0,Y 284.828,Z 239.002,A -85,B 0,C 180,E1 -17101.406,E2 -17101.406} C_VEL
LIN {X 0,Y 284.626,Z 239.03,A -85,B 0,C 180,E1 -17107.083,E2 -17107.083} C_VEL
LIN {X 0,Y 284.499,Z 239.042,A -85,B 0,C 180,E1 -17109.949,E2 -17109.949} C_VEL
LIN {X 0,Y 284.444,Z 239.051,A -85,B 0,C 180,E1 -17114.296,E2 -17114.296} C_VEL
LIN {X 0,Y 284.364,Z 239.056,A -85,B 0,C 180,E1 -17118.731,E2 -17118.731} C_VEL
LIN {X 0,Y 284.3,Z 239.07,A -85,B 0,C 180,E1 -17121.755,E2 -17121.755} C_VEL
LIN {X 0,Y 284.296,Z 239.069,A -85,B 0,C 180,E1 -17124.84,E2 -17124.84} C_VEL
LIN {X 0,Y 284.283,Z 239.064,A -85,B 0,C 180,E1 -17128.005,E2 -17128.005} C_VEL
LIN {X 0,Y 284.257,Z 239.061,A -85,B 0,C 180,E1 -17131.268,E2 -17131.268} C_VEL
LIN {X 0,Y 284.303,Z 239.066,A -85,B 0,C 180,E1 -17135.339,E2 -17135.339} C_VEL
LIN {X 0,Y 284.268,Z 239.072,A -85,B 0,C 180,E1 -17138.163,E2 -17138.163} C_VEL
LIN {X 0,Y 284.23,Z 239.076,A -85,B 0,C 180,E1 -17142.117,E2 -17142.117} C_VEL
LIN {X 0,Y 284.227,Z 239.078,A -85,B 0,C 180,E1 -17146.185,E2 -17146.185} C_VEL
LIN {X 0,Y 284.263,Z 239.071,A -85,B 0,C 180,E1 -17150.018,E2 -17150.018} C_VEL
LIN {X 0,Y 284.285,Z 239.073,A -85,B 0,C 180,E1 -17153.608,E2 -17153.608} C_VEL
LIN {X 0,Y 284.26,Z 239.077,A -85,B 0,C 180,E1 -17157.185,E2 -17157.185} C_VEL
LIN {X 0,Y 284.309,Z 239.069,A -85,B 0,C 180,E1 -17160.371,E2 -17160.371} C_VEL
LIN {X 0,Y 284.332,Z 239.068,A -85,B 0,C 180,E1 -17163.583,E2 -17163.583} C_VEL
LIN {X 0,Y 284.343,Z 239.067,A -85,B 0,C 180,E1 -17166.706,E2 -17166.706} C_VEL
LIN {X 0,Y 284.379,Z 239.062,A -85,B 0,C 180,E1 -17169.87,E2 -17169.87} C_VEL
LIN {X 0,Y 284.424,Z 239.056,A -85,B 0,C 180,E1 -17174.467,E2 -17174.467} C_VEL
LIN {X 0,Y 284.433,Z 239.054,A -85,B 0,C 180,E1 -17178.599,E2 -17178.599} C_VEL
LIN {X 0,Y 284.604,Z 239.033,A -85,B 0,C 180,E1 -17181.48,E2 -17181.48} C_VEL
LIN {X 0,Y 284.55,Z 239.038,A -85,B 0,C 180,E1 -17184.33,E2 -17184.33} C_VEL
LIN {X 0,Y 284.804,Z 239.008,A -85,B 0,C 180,E1 -17188.586,E2 -17188.586} C_VEL
LIN {X 0,Y 284.804,Z 239.008,A -85,B 0,C 180,E1 -17191.414,E2 -17191.414} C_VEL
LIN {X 0,Y 284.524,Z 239.203,A -85,B 0,C 180,E1 -17194.959,E2 -17194.959} C_VEL
LIN {X 0,Y 285.125,Z 241.648,A -85,B 0,C 180,E1 -17195.835,E2 -17195.835} C_VEL
LIN {X 0,Y 292.391,Z 261.015,A -85,B 0,C 180,E1 -17197.008,E2 -17197.008} C_VEL
LIN {X 0,Y 296.228,Z 272.442,A -85,B 0,C 180,E1 -17197.632,E2 -17197.632} C_VEL
LIN {X 0,Y 296.534,Z 275.069,A -85,B 0,C 180,E1 -17197.728,E2 -17197.728} C_VEL
LIN {X 0,Y 294.262,Z 349.709,A -85,B 0,C 180,E1 -17199.657,E2 -17199.657} C_VEL
LIN {X 0,Y 293.438,Z 363.228,A -85,B 0,C 180,E1 -17200.29,E2 -17200.29} C_VEL
LIN {X 0,Y 292.503,Z 375.833,A -85,B 0,C 180,E1 -17201.169,E2 -17201.169} C_VEL
LIN {X 0,Y 291.199,Z 388.453,A -85,B 0,C 180,E1 -17202.368,E2 -17202.368} C_VEL
LIN {X 0,Y 289.728,Z 400.21,A -85,B 0,C 180,E1 -17203.814,E2 -17203.814} C_VEL
LIN {X 0,Y 288.17,Z 411.263,A -85,B 0,C 180,E1 -17205.561,E2 -17205.561} C_VEL
LIN {X 0,Y 286.69,Z 420.778,A -85,B 0,C 180,E1 -17207.438,E2 -17207.438} C_VEL
LIN {X 0,Y 285.483,Z 428.767,A -85,B 0,C 180,E1 -17209.41,E2 -17209.41} C_VEL
LIN {X 0,Y 284.279,Z 436.351,A -85,B 0,C 180,E1 -17211.766,E2 -17211.766} C_VEL
LIN {X 0,Y 283.4,Z 442.398,A -85,B 0,C 180,E1 -17214.194,E2 -17214.194} C_VEL
LIN {X 0,Y 282.918,Z 446.85,A -85,B 0,C 180,E1 -17216.609,E2 -17216.609} C_VEL
LIN {X 0,Y 282.596,Z 449.069,A -85,B 0,C 180,E1 -17218.197,E2 -17218.197} C_VEL
LIN {X 0,Y 282.273,Z 450.811,A -85,B 0,C 180,E1 -17219.864,E2 -17219.864} C_VEL
LIN {X 0,Y 282.092,Z 452.267,A -85,B 0,C 180,E1 -17222.126,E2 -17222.126} C_VEL
LIN {X 0,Y 282.169,Z 452.664,A -85,B 0,C 180,E1 -17224.949,E2 -17224.949} C_VEL
LIN {X 0,Y 282.462,Z 451.833,A -85,B 0,C 180,E1 -17227.249,E2 -17227.249} C_VEL
LIN {X 0,Y 283.007,Z 449.824,A -85,B 0,C 180,E1 -17229.678,E2 -17229.678} C_VEL
LIN {X 0,Y 283.742,Z 446.711,A -85,B 0,C 180,E1 -17232.022,E2 -17232.022} C_VEL
LIN {X 0,Y 284.743,Z 442.441,A -85,B 0,C 180,E1 -17234.308,E2 -17234.308} C_VEL
LIN {X 0,Y 286.238,Z 435.959,A -85,B 0,C 180,E1 -17236.89,E2 -17236.89} C_VEL
LIN {X 0,Y 287.954,Z 428.518,A -85,B 0,C 180,E1 -17239.164,E2 -17239.164} C_VEL
LIN {X 0,Y 289.822,Z 420.155,A -85,B 0,C 180,E1 -17241.168,E2 -17241.168} C_VEL
LIN {X 0,Y 291.807,Z 410.697,A -85,B 0,C 180,E1 -17242.991,E2 -17242.991} C_VEL
LIN {X 0,Y 293.611,Z 401.174,A -85,B 0,C 180,E1 -17244.471,E2 -17244.471} C_VEL
LIN {X 0,Y 295.422,Z 389.965,A -85,B 0,C 180,E1 -17245.857,E2 -17245.857} C_VEL
LIN {X 0,Y 297.102,Z 377.483,A -85,B 0,C 180,E1 -17247.05,E2 -17247.05} C_VEL
LIN {X 0,Y 298.358,Z 365.743,A -85,B 0,C 180,E1 -17247.886,E2 -17247.886} C_VEL
LIN {X 0,Y 299.326,Z 353.062,A -85,B 0,C 180,E1 -17248.512,E2 -17248.512} C_VEL
LIN {X 0,Y 300.096,Z 334.78,A -85,B 0,C 180,E1 -17249.048,E2 -17249.048} C_VEL
LIN {X 0,Y 302.161,Z 277.865,A -85,B 0,C 180,E1 -17250.508,E2 -17250.508} C_VEL
LIN {X 0,Y 297.909,Z 267.661,A -85,B 0,C 180,E1 -17251.343,E2 -17251.343} C_VEL
LIN {X 0,Y 295.502,Z 262.797,A -85,B 0,C 180,E1 -17251.807,E2 -17251.807} C_VEL
LIN {X 0,Y 292.471,Z 258.493,A -85,B 0,C 180,E1 -17252.349,E2 -17252.349} C_VEL
LIN {X 0,Y 290.217,Z 255.902,A -85,B 0,C 180,E1 -17252.743,E2 -17252.743} C_VEL
LIN {X 0,Y 285.317,Z 251.168,A -85,B 0,C 180,E1 -17253.602,E2 -17253.602} C_VEL
LIN {X 0,Y 280.247,Z 246.821,A -85,B 0,C 180,E1 -17254.522,E2 -17254.522} C_VEL
LIN {X 0,Y 278.16,Z 242.977,A -85,B 0,C 180,E1 -17255.044,E2 -17255.044} C_VEL
LIN {X 0,Y 277.309,Z 239.943,A -85,B 0,C 180,E1 -17256.386,E2 -17256.386} C_VEL
LIN {X 0,Y 277.323,Z 239.942,A -85,B 0,C 180,E1 -17260.775,E2 -17260.775} C_VEL
LIN {X 0,Y 277.41,Z 239.926,A -85,B 0,C 180,E1 -17265.334,E2 -17265.334} C_VEL
LIN {X 0,Y 277.445,Z 239.926,A -85,B 0,C 180,E1 -17269.795,E2 -17269.795} C_VEL
LIN {X 0,Y 277.608,Z 239.904,A -85,B 0,C 180,E1 -17272.737,E2 -17272.737} C_VEL
LIN {X 0,Y 277.809,Z 239.872,A -85,B 0,C 180,E1 -17278.559,E2 -17278.559} C_VEL
LIN {X 0,Y 277.805,Z 239.873,A -85,B 0,C 180,E1 -17281.458,E2 -17281.458} C_VEL
LIN {X 0,Y 277.611,Z 239.901,A -85,B 0,C 180,E1 -17287.28,E2 -17287.28} C_VEL
LIN {X 0,Y 277.456,Z 239.913,A -85,B 0,C 180,E1 -17290.221,E2 -17290.221} C_VEL
LIN {X 0,Y 277.41,Z 239.92,A -85,B 0,C 180,E1 -17294.683,E2 -17294.683} C_VEL
LIN {X 0,Y 277.287,Z 239.938,A -85,B 0,C 180,E1 -17299.245,E2 -17299.245} C_VEL
LIN {X 0,Y 277.263,Z 239.944,A -85,B 0,C 180,E1 -17303.934,E2 -17303.934} C_VEL
LIN {X 0,Y 277.242,Z 239.947,A -85,B 0,C 180,E1 -17307.475,E2 -17307.475} C_VEL
LIN {X 0,Y 277.238,Z 239.943,A -85,B 0,C 180,E1 -17310.472,E2 -17310.472} C_VEL
LIN {X 0,Y 277.249,Z 239.942,A -85,B 0,C 180,E1 -17313.903,E2 -17313.903} C_VEL
LIN {X 0,Y 277.241,Z 239.948,A -85,B 0,C 180,E1 -17317.481,E2 -17317.481} C_VEL
LIN {X 0,Y 277.175,Z 239.962,A -85,B 0,C 180,E1 -17321.251,E2 -17321.251} C_VEL
LIN {X 0,Y 277.179,Z 239.961,A -85,B 0,C 180,E1 -17325.239,E2 -17325.239} C_VEL
LIN {X 0,Y 277.186,Z 239.96,A -85,B 0,C 180,E1 -17329.53,E2 -17329.53} C_VEL
LIN {X 0,Y 277.241,Z 240.095,A -85,B 0,C 180,E1 -17331.462,E2 -17331.462} C_VEL
LIN {X 0,Y 279.525,Z 247.939,A -85,B 0,C 180,E1 -17334.672,E2 -17334.672} C_VEL
LIN {X 0,Y 282.084,Z 258.738,A -85,B 0,C 180,E1 -17338.673,E2 -17338.673} C_VEL
LIN {X 0,Y 289.662,Z 275.601,A -85,B 0,C 180,E1 -17340.324,E2 -17340.324} C_VEL
LIN {X 0,Y 290.819,Z 280.111,A -85,B 0,C 180,E1 -17340.625,E2 -17340.625} C_VEL
LIN {X 0,Y 294.135,Z 300.253,A -85,B 0,C 180,E1 -17341.694,E2 -17341.694} C_VEL
LIN {X 0,Y 295.127,Z 309.198,A -85,B 0,C 180,E1 -17342.097,E2 -17342.097} C_VEL
LIN {X 0,Y 292.842,Z 368.802,A -85,B 0,C 180,E1 -17343.69,E2 -17343.69} C_VEL
LIN {X 0,Y 291.582,Z 382.927,A -85,B 0,C 180,E1 -17344.336,E2 -17344.336} C_VEL
LIN {X 0,Y 290.034,Z 395.491,A -85,B 0,C 180,E1 -17345.197,E2 -17345.197} C_VEL
LIN {X 0,Y 288.142,Z 407.125,A -85,B 0,C 180,E1 -17346.269,E2 -17346.269} C_VEL
LIN {X 0,Y 286.148,Z 418.407,A -85,B 0,C 180,E1 -17347.624,E2 -17347.624} C_VEL
LIN {X 0,Y 284.07,Z 428.643,A -85,B 0,C 180,E1 -17349.168,E2 -17349.168} C_VEL
LIN {X 0,Y 281.844,Z 438.696,A -85,B 0,C 180,E1 -17351.086,E2 -17351.086} C_VEL
LIN {X 0,Y 279.919,Z 447.576,A -85,B 0,C 180,E1 -17353.218,E2 -17353.218} C_VEL
LIN {X 0,Y 278.3,Z 454.731,A -85,B 0,C 180,E1 -17355.373,E2 -17355.373} C_VEL
LIN {X 0,Y 276.968,Z 460.478,A -85,B 0,C 180,E1 -17357.545,E2 -17357.545} C_VEL
LIN {X 0,Y 276.15,Z 465.028,A -85,B 0,C 180,E1 -17359.738,E2 -17359.738} C_VEL
LIN {X 0,Y 275.74,Z 467.442,A -85,B 0,C 180,E1 -17361.204,E2 -17361.204} C_VEL
LIN {X 0,Y 275.468,Z 469.428,A -85,B 0,C 180,E1 -17362.671,E2 -17362.671} C_VEL
LIN {X 0,Y 275.29,Z 471.445,A -85,B 0,C 180,E1 -17364.705,E2 -17364.705} C_VEL
LIN {X 0,Y 275.288,Z 472.809,A -85,B 0,C 180,E1 -17367.073,E2 -17367.073} C_VEL
LIN {X 0,Y 275.295,Z 473.132,A -85,B 0,C 180,E1 -17368.537,E2 -17368.537} C_VEL
LIN {X 0,Y 275.322,Z 473.048,A -85,B 0,C 180,E1 -17370,E2 -17370} C_VEL
LIN {X 0,Y 275.304,Z 472.519,A -85,B 0,C 180,E1 -17371.463,E2 -17371.463} C_VEL
LIN {X 0,Y 275.298,Z 471.588,A -85,B 0,C 180,E1 -17372.927,E2 -17372.927} C_VEL
LIN {X 0,Y 275.334,Z 469.065,A -85,B 0,C 180,E1 -17375.394,E2 -17375.394} C_VEL
LIN {X 0,Y 275.589,Z 464.9,A -85,B 0,C 180,E1 -17378.063,E2 -17378.063} C_VEL
LIN {X 0,Y 276.052,Z 460.197,A -85,B 0,C 180,E1 -17380.265,E2 -17380.265} C_VEL
LIN {X 0,Y 276.949,Z 453.077,A -85,B 0,C 180,E1 -17382.829,E2 -17382.829} C_VEL
LIN {X 0,Y 278.162,Z 445.354,A -85,B 0,C 180,E1 -17385.009,E2 -17385.009} C_VEL
LIN {X 0,Y 279.538,Z 436.488,A -85,B 0,C 180,E1 -17387,E2 -17387} C_VEL
LIN {X 0,Y 280.978,Z 426.637,A -85,B 0,C 180,E1 -17388.786,E2 -17388.786} C_VEL
LIN {X 0,Y 282.606,Z 415.634,A -85,B 0,C 180,E1 -17390.374,E2 -17390.374} C_VEL
LIN {X 0,Y 284.274,Z 403.098,A -85,B 0,C 180,E1 -17391.767,E2 -17391.767} C_VEL
LIN {X 0,Y 285.661,Z 390.826,A -85,B 0,C 180,E1 -17392.798,E2 -17392.798} C_VEL
LIN {X 0,Y 286.751,Z 377.953,A -85,B 0,C 180,E1 -17393.565,E2 -17393.565} C_VEL
LIN {X 0,Y 287.518,Z 364.603,A -85,B 0,C 180,E1 -17394.073,E2 -17394.073} C_VEL
LIN {X 0,Y 289.057,Z 305.991,A -85,B 0,C 180,E1 -17395.616,E2 -17395.616} C_VEL
LIN {X 0,Y 283.487,Z 267.096,A -85,B 0,C 180,E1 -17397.196,E2 -17397.196} C_VEL
LIN {X 0,Y 281.631,Z 260.848,A -85,B 0,C 180,E1 -17397.569,E2 -17397.569} C_VEL
LIN {X 0,Y 279.248,Z 248.979,A -85,B 0,C 180,E1 -17401.455,E2 -17401.455} C_VEL
LIN {X 0,Y 277.285,Z 239.946,A -85,B 0,C 180,E1 -17404.603,E2 -17404.603} C_VEL
LIN {X 0,Y 277.237,Z 239.949,A -85,B 0,C 180,E1 -17408.191,E2 -17408.191} C_VEL
LIN {X 0,Y 277.159,Z 239.96,A -85,B 0,C 180,E1 -17412.654,E2 -17412.654} C_VEL
LIN {X 0,Y 277.162,Z 239.96,A -85,B 0,C 180,E1 -17416.785,E2 -17416.785} C_VEL
LIN {X 0,Y 277.203,Z 239.953,A -85,B 0,C 180,E1 -17420.659,E2 -17420.659} C_VEL
LIN {X 0,Y 277.286,Z 239.944,A -85,B 0,C 180,E1 -17424.334,E2 -17424.334} C_VEL
LIN {X 0,Y 277.235,Z 239.952,A -85,B 0,C 180,E1 -17427.828,E2 -17427.828} C_VEL
LIN {X 0,Y 277.222,Z 239.953,A -85,B 0,C 180,E1 -17431.197,E2 -17431.197} C_VEL
LIN {X 0,Y 277.241,Z 239.948,A -85,B 0,C 180,E1 -17434.465,E2 -17434.465} C_VEL
LIN {X 0,Y 277.253,Z 239.949,A -85,B 0,C 180,E1 -17437.645,E2 -17437.645} C_VEL
LIN {X 0,Y 277.282,Z 239.935,A -85,B 0,C 180,E1 -17440.754,E2 -17440.754} C_VEL
LIN {X 0,Y 277.41,Z 239.924,A -85,B 0,C 180,E1 -17445.317,E2 -17445.317} C_VEL
LIN {X 0,Y 277.451,Z 239.924,A -85,B 0,C 180,E1 -17449.779,E2 -17449.779} C_VEL
LIN {X 0,Y 277.587,Z 239.9,A -85,B 0,C 180,E1 -17452.72,E2 -17452.72} C_VEL
LIN {X 0,Y 277.796,Z 239.867,A -85,B 0,C 180,E1 -17458.542,E2 -17458.542} C_VEL
LIN {X 0,Y 277.795,Z 239.878,A -85,B 0,C 180,E1 -17461.441,E2 -17461.441} C_VEL
LIN {X 0,Y 277.585,Z 239.908,A -85,B 0,C 180,E1 -17467.264,E2 -17467.264} C_VEL
LIN {X 0,Y 277.442,Z 239.92,A -85,B 0,C 180,E1 -17470.205,E2 -17470.205} C_VEL
LIN {X 0,Y 277.391,Z 239.929,A -85,B 0,C 180,E1 -17474.667,E2 -17474.667} C_VEL
LIN {X 0,Y 277.313,Z 239.937,A -85,B 0,C 180,E1 -17479.226,E2 -17479.226} C_VEL
LIN {X 0,Y 277.265,Z 239.945,A -85,B 0,C 180,E1 -17483.916,E2 -17483.916} C_VEL
LIN {X 0,Y 277.28,Z 239.939,A -85,B 0,C 180,E1 -17487.489,E2 -17487.489} C_VEL
LIN {X 0,Y 277.218,Z 239.935,A -85,B 0,C 180,E1 -17490.465,E2 -17490.465} C_VEL
LIN {X 0,Y 277.213,Z 239.944,A -85,B 0,C 180,E1 -17493.888,E2 -17493.888} C_VEL
LIN {X 0,Y 277.223,Z 239.953,A -85,B 0,C 180,E1 -17497.463,E2 -17497.463} C_VEL
LIN {X 0,Y 277.172,Z 239.961,A -85,B 0,C 180,E1 -17501.229,E2 -17501.229} C_VEL
LIN {X 0,Y 277.172,Z 239.959,A -85,B 0,C 180,E1 -17505.217,E2 -17505.217} C_VEL
LIN {X 0,Y 277.179,Z 239.955,A -85,B 0,C 180,E1 -17509.506,E2 -17509.506} C_VEL
LIN {X 0,Y 277.221,Z 239.951,A -85,B 0,C 180,E1 -17512.524,E2 -17512.524} C_VEL
LIN {X 0,Y 277.2,Z 239.952,A -85,B 0,C 180,E1 -17516.099,E2 -17516.099} C_VEL
LIN {X 0,Y 277.214,Z 239.955,A -85,B 0,C 180,E1 -17519.534,E2 -17519.534} C_VEL
LIN {X 0,Y 277.311,Z 239.941,A -85,B 0,C 180,E1 -17522.86,E2 -17522.86} C_VEL
LIN {X 0,Y 277.326,Z 239.94,A -85,B 0,C 180,E1 -17526.08,E2 -17526.08} C_VEL
LIN {X 0,Y 277.318,Z 239.943,A -85,B 0,C 180,E1 -17530.765,E2 -17530.765} C_VEL
LIN {X 0,Y 277.373,Z 239.934,A -85,B 0,C 180,E1 -17535.323,E2 -17535.323} C_VEL
LIN {X 0,Y 277.451,Z 239.922,A -85,B 0,C 180,E1 -17539.787,E2 -17539.787} C_VEL
LIN {X 0,Y 277.599,Z 239.905,A -85,B 0,C 180,E1 -17542.728,E2 -17542.728} C_VEL
LIN {X 0,Y 277.77,Z 239.885,A -85,B 0,C 180,E1 -17548.55,E2 -17548.55} C_VEL
LIN {X 0,Y 277.77,Z 239.884,A -85,B 0,C 180,E1 -17551.45,E2 -17551.45} C_VEL
LIN {X 0,Y 277.478,Z 240.121,A -85,B 0,C 180,E1 -17554.54,E2 -17554.54} C_VEL
LIN {X 0,Y 277.857,Z 241.827,A -85,B 0,C 180,E1 -17555.17,E2 -17555.17} C_VEL
LIN {X 0,Y 284.306,Z 258.257,A -85,B 0,C 180,E1 -17556.252,E2 -17556.252} C_VEL
LIN {X 0,Y 289.847,Z 274.663,A -85,B 0,C 180,E1 -17557.189,E2 -17557.189} C_VEL
LIN {X 0,Y 287.59,Z 349.82,A -85,B 0,C 180,E1 -17559.184,E2 -17559.184} C_VEL
LIN {X 0,Y 286.757,Z 362.713,A -85,B 0,C 180,E1 -17559.789,E2 -17559.789} C_VEL
LIN {X 0,Y 285.831,Z 374.967,A -85,B 0,C 180,E1 -17560.641,E2 -17560.641} C_VEL
LIN {X 0,Y 284.597,Z 386.866,A -85,B 0,C 180,E1 -17561.755,E2 -17561.755} C_VEL
LIN {X 0,Y 283.123,Z 398.847,A -85,B 0,C 180,E1 -17563.217,E2 -17563.217} C_VEL
LIN {X 0,Y 281.609,Z 409.274,A -85,B 0,C 180,E1 -17564.821,E2 -17564.821} C_VEL
LIN {X 0,Y 279.99,Z 419.248,A -85,B 0,C 180,E1 -17566.755,E2 -17566.755} C_VEL
LIN {X 0,Y 278.727,Z 427.514,A -85,B 0,C 180,E1 -17568.752,E2 -17568.752} C_VEL
LIN {X 0,Y 277.652,Z 434.236,A -85,B 0,C 180,E1 -17570.754,E2 -17570.754} C_VEL
LIN {X 0,Y 276.691,Z 440.45,A -85,B 0,C 180,E1 -17573.079,E2 -17573.079} C_VEL
LIN {X 0,Y 275.974,Z 445.657,A -85,B 0,C 180,E1 -17575.652,E2 -17575.652} C_VEL
LIN {X 0,Y 275.759,Z 448.236,A -85,B 0,C 180,E1 -17577.305,E2 -17577.305} C_VEL
LIN {X 0,Y 275.189,Z 450.978,A -85,B 0,C 180,E1 -17579.759,E2 -17579.759} C_VEL
LIN {X 0,Y 274.992,Z 452.646,A -85,B 0,C 180,E1 -17582.522,E2 -17582.522} C_VEL
LIN {X 0,Y 275.091,Z 452.925,A -85,B 0,C 180,E1 -17585.181,E2 -17585.181} C_VEL
LIN {X 0,Y 275.453,Z 451.94,A -85,B 0,C 180,E1 -17587.758,E2 -17587.758} C_VEL
LIN {X 0,Y 276.077,Z 449.79,A -85,B 0,C 180,E1 -17590.225,E2 -17590.225} C_VEL
LIN {X 0,Y 276.885,Z 446.538,A -85,B 0,C 180,E1 -17592.617,E2 -17592.617} C_VEL
LIN {X 0,Y 278.049,Z 441.919,A -85,B 0,C 180,E1 -17595.049,E2 -17595.049} C_VEL
LIN {X 0,Y 279.375,Z 436.515,A -85,B 0,C 180,E1 -17597.232,E2 -17597.232} C_VEL
LIN {X 0,Y 281.078,Z 429.51,A -85,B 0,C 180,E1 -17599.465,E2 -17599.465} C_VEL
LIN {X 0,Y 282.903,Z 421.998,A -85,B 0,C 180,E1 -17601.37,E2 -17601.37} C_VEL
LIN {X 0,Y 284.961,Z 412.637,A -85,B 0,C 180,E1 -17603.276,E2 -17603.276} C_VEL
LIN {X 0,Y 286.866,Z 403.055,A -85,B 0,C 180,E1 -17604.849,E2 -17604.849} C_VEL
LIN {X 0,Y 288.688,Z 393.012,A -85,B 0,C 180,E1 -17606.174,E2 -17606.174} C_VEL
LIN {X 0,Y 290.402,Z 381.307,A -85,B 0,C 180,E1 -17607.402,E2 -17607.402} C_VEL
LIN {X 0,Y 291.857,Z 369.152,A -85,B 0,C 180,E1 -17608.353,E2 -17608.353} C_VEL
LIN {X 0,Y 292.992,Z 355.989,A -85,B 0,C 180,E1 -17609.089,E2 -17609.089} C_VEL
LIN {X 0,Y 293.704,Z 342.299,A -85,B 0,C 180,E1 -17609.555,E2 -17609.555} C_VEL
LIN {X 0,Y 296.096,Z 279.72,A -85,B 0,C 180,E1 -17611.198,E2 -17611.198} C_VEL
LIN {X 0,Y 289.7,Z 264.863,A -85,B 0,C 180,E1 -17612.517,E2 -17612.517} C_VEL
LIN {X 0,Y 283.684,Z 253.132,A -85,B 0,C 180,E1 -17613.775,E2 -17613.775} C_VEL
LIN {X 0,Y 280.247,Z 246.821,A -85,B 0,C 180,E1 -17614.522,E2 -17614.522} C_VEL
LIN {X 0,Y 276.759,Z 244.263,A -85,B 0,C 180,E1 -17615.243,E2 -17615.243} C_VEL
LIN {X 0,Y 273.216,Z 242.269,A -85,B 0,C 180,E1 -17616.227,E2 -17616.227} C_VEL
LIN {X 0,Y 270.784,Z 241.071,A -85,B 0,C 180,E1 -17617.379,E2 -17617.379} C_VEL
LIN {X 0,Y 270.2,Z 240.828,A -85,B 0,C 180,E1 -17618.223,E2 -17618.223} C_VEL
LIN {X 0,Y 270.269,Z 240.822,A -85,B 0,C 180,E1 -17621.828,E2 -17621.828} C_VEL
LIN {X 0,Y 270.378,Z 240.804,A -85,B 0,C 180,E1 -17624.944,E2 -17624.944} C_VEL
LIN {X 0,Y 270.398,Z 240.805,A -85,B 0,C 180,E1 -17629.526,E2 -17629.526} C_VEL
LIN {X 0,Y 270.565,Z 240.78,A -85,B 0,C 180,E1 -17632.547,E2 -17632.547} C_VEL
LIN {X 0,Y 270.775,Z 240.748,A -85,B 0,C 180,E1 -17638.521,E2 -17638.521} C_VEL
LIN {X 0,Y 270.77,Z 240.749,A -85,B 0,C 180,E1 -17641.496,E2 -17641.496} C_VEL
LIN {X 0,Y 270.571,Z 240.78,A -85,B 0,C 180,E1 -17647.47,E2 -17647.47} C_VEL
LIN {X 0,Y 270.408,Z 240.791,A -85,B 0,C 180,E1 -17650.49,E2 -17650.49} C_VEL
LIN {X 0,Y 270.369,Z 240.8,A -85,B 0,C 180,E1 -17655.074,E2 -17655.074} C_VEL
LIN {X 0,Y 270.227,Z 240.821,A -85,B 0,C 180,E1 -17659.769,E2 -17659.769} C_VEL
LIN {X 0,Y 270.189,Z 240.829,A -85,B 0,C 180,E1 -17664.443,E2 -17664.443} C_VEL
LIN {X 0,Y 270.192,Z 240.826,A -85,B 0,C 180,E1 -17667.925,E2 -17667.925} C_VEL
LIN {X 0,Y 270.174,Z 240.83,A -85,B 0,C 180,E1 -17671.357,E2 -17671.357} C_VEL
LIN {X 0,Y 270.205,Z 240.828,A -85,B 0,C 180,E1 -17674.913,E2 -17674.913} C_VEL
LIN {X 0,Y 270.181,Z 240.83,A -85,B 0,C 180,E1 -17678.708,E2 -17678.708} C_VEL
LIN {X 0,Y 270.128,Z 240.84,A -85,B 0,C 180,E1 -17683.242,E2 -17683.242} C_VEL
LIN {X 0,Y 270.132,Z 240.839,A -85,B 0,C 180,E1 -17687.436,E2 -17687.436} C_VEL
LIN {X 0,Y 270.174,Z 240.954,A -85,B 0,C 180,E1 -17690.41,E2 -17690.41} C_VEL
LIN {X 0,Y 272.733,Z 249.567,A -85,B 0,C 180,E1 -17694.111,E2 -17694.111} C_VEL
LIN {X 0,Y 274.901,Z 258.606,A -85,B 0,C 180,E1 -17697.539,E2 -17697.539} C_VEL
LIN {X 0,Y 281.33,Z 272.123,A -85,B 0,C 180,E1 -17699.019,E2 -17699.019} C_VEL
LIN {X 0,Y 284.689,Z 280.146,A -85,B 0,C 180,E1 -17699.782,E2 -17699.782} C_VEL
LIN {X 0,Y 288.197,Z 301.442,A -85,B 0,C 180,E1 -17700.96,E2 -17700.96} C_VEL
LIN {X 0,Y 289.105,Z 310.375,A -85,B 0,C 180,E1 -17701.367,E2 -17701.367} C_VEL
LIN {X 0,Y 286.809,Z 368.039,A -85,B 0,C 180,E1 -17702.945,E2 -17702.945} C_VEL
LIN {X 0,Y 285.563,Z 381.535,A -85,B 0,C 180,E1 -17703.558,E2 -17703.558} C_VEL
LIN {X 0,Y 283.95,Z 394.411,A -85,B 0,C 180,E1 -17704.432,E2 -17704.432} C_VEL
LIN {X 0,Y 281.96,Z 406.212,A -85,B 0,C 180,E1 -17705.52,E2 -17705.52} C_VEL
LIN {X 0,Y 279.878,Z 417.609,A -85,B 0,C 180,E1 -17706.899,E2 -17706.899} C_VEL
LIN {X 0,Y 277.66,Z 427.947,A -85,B 0,C 180,E1 -17708.469,E2 -17708.469} C_VEL
LIN {X 0,Y 275.526,Z 437.275,A -85,B 0,C 180,E1 -17710.247,E2 -17710.247} C_VEL
LIN {X 0,Y 273.456,Z 446.347,A -85,B 0,C 180,E1 -17712.424,E2 -17712.424} C_VEL
LIN {X 0,Y 271.711,Z 453.691,A -85,B 0,C 180,E1 -17714.626,E2 -17714.626} C_VEL
LIN {X 0,Y 270.396,Z 458.682,A -85,B 0,C 180,E1 -17716.472,E2 -17716.472} C_VEL
LIN {X 0,Y 269.376,Z 463.554,A -85,B 0,C 180,E1 -17718.716,E2 -17718.716} C_VEL
LIN {X 0,Y 268.703,Z 467.317,A -85,B 0,C 180,E1 -17720.972,E2 -17720.972} C_VEL
LIN {X 0,Y 268.392,Z 469.281,A -85,B 0,C 180,E1 -17722.477,E2 -17722.477} C_VEL
LIN {X 0,Y 268.186,Z 471.45,A -85,B 0,C 180,E1 -17724.813,E2 -17724.813} C_VEL
LIN {X 0,Y 268.197,Z 472.577,A -85,B 0,C 180,E1 -17726.996,E2 -17726.996} C_VEL
LIN {X 0,Y 268.22,Z 472.879,A -85,B 0,C 180,E1 -17728.499,E2 -17728.499} C_VEL
LIN {X 0,Y 268.245,Z 472.754,A -85,B 0,C 180,E1 -17730,E2 -17730} C_VEL
LIN {X 0,Y 268.229,Z 472.201,A -85,B 0,C 180,E1 -17731.501,E2 -17731.501} C_VEL
LIN {X 0,Y 268.208,Z 471.246,A -85,B 0,C 180,E1 -17733.004,E2 -17733.004} C_VEL
LIN {X 0,Y 268.228,Z 468.978,A -85,B 0,C 180,E1 -17735.284,E2 -17735.284} C_VEL
LIN {X 0,Y 268.424,Z 465.747,A -85,B 0,C 180,E1 -17737.522,E2 -17737.522} C_VEL
LIN {X 0,Y 268.831,Z 461.385,A -85,B 0,C 180,E1 -17739.783,E2 -17739.783} C_VEL
LIN {X 0,Y 269.476,Z 455.796,A -85,B 0,C 180,E1 -17742.043,E2 -17742.043} C_VEL
LIN {X 0,Y 270.651,Z 448.813,A -85,B 0,C 180,E1 -17744.281,E2 -17744.281} C_VEL
LIN {X 0,Y 271.835,Z 441.66,A -85,B 0,C 180,E1 -17746.136,E2 -17746.136} C_VEL
LIN {X 0,Y 273.115,Z 432.977,A -85,B 0,C 180,E1 -17747.986,E2 -17747.986} C_VEL
LIN {X 0,Y 274.791,Z 422.279,A -85,B 0,C 180,E1 -17749.808,E2 -17749.808} C_VEL
LIN {X 0,Y 276.339,Z 411.677,A -85,B 0,C 180,E1 -17751.248,E2 -17751.248} C_VEL
LIN {X 0,Y 277.89,Z 399.941,A -85,B 0,C 180,E1 -17752.489,E2 -17752.489} C_VEL
LIN {X 0,Y 279.377,Z 386.535,A -85,B 0,C 180,E1 -17753.537,E2 -17753.537} C_VEL
LIN {X 0,Y 280.362,Z 373.765,A -85,B 0,C 180,E1 -17754.235,E2 -17754.235} C_VEL
LIN {X 0,Y 281.038,Z 358.976,A -85,B 0,C 180,E1 -17754.713,E2 -17754.713} C_VEL
LIN {X 0,Y 282.423,Z 306.922,A -85,B 0,C 180,E1 -17756.115,E2 -17756.115} C_VEL
LIN {X 0,Y 277.106,Z 268.988,A -85,B 0,C 180,E1 -17757.7,E2 -17757.7} C_VEL
LIN {X 0,Y 274.359,Z 260.577,A -85,B 0,C 180,E1 -17758.23,E2 -17758.23} C_VEL
LIN {X 0,Y 272.343,Z 250.562,A -85,B 0,C 180,E1 -17761.605,E2 -17761.605} C_VEL
LIN {X 0,Y 270.239,Z 240.824,A -85,B 0,C 180,E1 -17765.07,E2 -17765.07} C_VEL
LIN {X 0,Y 270.186,Z 240.826,A -85,B 0,C 180,E1 -17768.698,E2 -17768.698} C_VEL
LIN {X 0,Y 270.116,Z 240.838,A -85,B 0,C 180,E1 -17773.229,E2 -17773.229} C_VEL
LIN {X 0,Y 270.129,Z 240.838,A -85,B 0,C 180,E1 -17777.425,E2 -17777.425} C_VEL
LIN {X 0,Y 270.165,Z 240.832,A -85,B 0,C 180,E1 -17781.359,E2 -17781.359} C_VEL
LIN {X 0,Y 270.205,Z 240.826,A -85,B 0,C 180,E1 -17785.087,E2 -17785.087} C_VEL
LIN {X 0,Y 270.18,Z 240.828,A -85,B 0,C 180,E1 -17789.136,E2 -17789.136} C_VEL
LIN {X 0,Y 270.196,Z 240.826,A -85,B 0,C 180,E1 -17792.171,E2 -17792.171} C_VEL
LIN {X 0,Y 270.191,Z 240.83,A -85,B 0,C 180,E1 -17795.556,E2 -17795.556} C_VEL
LIN {X 0,Y 270.225,Z 240.814,A -85,B 0,C 180,E1 -17800.231,E2 -17800.231} C_VEL
LIN {X 0,Y 270.369,Z 240.798,A -85,B 0,C 180,E1 -17804.926,E2 -17804.926} C_VEL
LIN {X 0,Y 270.385,Z 240.807,A -85,B 0,C 180,E1 -17809.509,E2 -17809.509} C_VEL
LIN {X 0,Y 270.549,Z 240.777,A -85,B 0,C 180,E1 -17812.529,E2 -17812.529} C_VEL
LIN {X 0,Y 270.759,Z 240.742,A -85,B 0,C 180,E1 -17818.504,E2 -17818.504} C_VEL
LIN {X 0,Y 270.761,Z 240.754,A -85,B 0,C 180,E1 -17821.479,E2 -17821.479} C_VEL
LIN {X 0,Y 270.547,Z 240.783,A -85,B 0,C 180,E1 -17827.454,E2 -17827.454} C_VEL
LIN {X 0,Y 270.395,Z 240.797,A -85,B 0,C 180,E1 -17830.474,E2 -17830.474} C_VEL
LIN {X 0,Y 270.359,Z 240.807,A -85,B 0,C 180,E1 -17835.057,E2 -17835.057} C_VEL
LIN {X 0,Y 270.275,Z 240.815,A -85,B 0,C 180,E1 -17839.747,E2 -17839.747} C_VEL
LIN {X 0,Y 270.208,Z 240.823,A -85,B 0,C 180,E1 -17844.581,E2 -17844.581} C_VEL
LIN {X 0,Y 270.215,Z 240.815,A -85,B 0,C 180,E1 -17847.904,E2 -17847.904} C_VEL
LIN {X 0,Y 270.143,Z 240.814,A -85,B 0,C 180,E1 -17851.341,E2 -17851.341} C_VEL
LIN {X 0,Y 270.165,Z 240.821,A -85,B 0,C 180,E1 -17854.898,E2 -17854.898} C_VEL
LIN {X 0,Y 270.162,Z 240.83,A -85,B 0,C 180,E1 -17858.703,E2 -17858.703} C_VEL
LIN {X 0,Y 270.127,Z 240.834,A -85,B 0,C 180,E1 -17863.242,E2 -17863.242} C_VEL
LIN {X 0,Y 270.132,Z 240.837,A -85,B 0,C 180,E1 -17867.435,E2 -17867.435} C_VEL
LIN {X 0,Y 270.164,Z 240.832,A -85,B 0,C 180,E1 -17871.368,E2 -17871.368} C_VEL
LIN {X 0,Y 270.155,Z 240.835,A -85,B 0,C 180,E1 -17875.089,E2 -17875.089} C_VEL
LIN {X 0,Y 270.153,Z 240.836,A -85,B 0,C 180,E1 -17879.126,E2 -17879.126} C_VEL
LIN {X 0,Y 270.216,Z 240.823,A -85,B 0,C 180,E1 -17882.141,E2 -17882.141} C_VEL
LIN {X 0,Y 270.264,Z 240.822,A -85,B 0,C 180,E1 -17885.498,E2 -17885.498} C_VEL
LIN {X 0,Y 270.275,Z 240.819,A -85,B 0,C 180,E1 -17890.243,E2 -17890.243} C_VEL
LIN {X 0,Y 270.342,Z 240.813,A -85,B 0,C 180,E1 -17894.932,E2 -17894.932} C_VEL
LIN {X 0,Y 270.387,Z 240.803,A -85,B 0,C 180,E1 -17899.517,E2 -17899.517} C_VEL
LIN {X 0,Y 270.557,Z 240.782,A -85,B 0,C 180,E1 -17902.537,E2 -17902.537} C_VEL
LIN {X 0,Y 270.736,Z 240.761,A -85,B 0,C 180,E1 -17908.512,E2 -17908.512} C_VEL
LIN {X 0,Y 270.736,Z 240.76,A -85,B 0,C 180,E1 -17911.487,E2 -17911.487} C_VEL
LIN {X 0,Y 270.446,Z 240.892,A -85,B 0,C 180,E1 -17914.051,E2 -17914.051} C_VEL
LIN {X 0,Y 270.687,Z 242.11,A -85,B 0,C 180,E1 -17914.509,E2 -17914.509} C_VEL
LIN {X 0,Y 277.856,Z 260.126,A -85,B 0,C 180,E1 -17915.738,E2 -17915.738} C_VEL
LIN {X 0,Y 283.369,Z 276.224,A -85,B 0,C 180,E1 -17916.698,E2 -17916.698} C_VEL
LIN {X 0,Y 280.96,Z 349.643,A -85,B 0,C 180,E1 -17918.677,E2 -17918.677} C_VEL
LIN {X 0,Y 280.052,Z 363.455,A -85,B 0,C 180,E1 -17919.342,E2 -17919.342} C_VEL
LIN {X 0,Y 279.046,Z 376.195,A -85,B 0,C 180,E1 -17920.266,E2 -17920.266} C_VEL
LIN {X 0,Y 277.656,Z 388.904,A -85,B 0,C 180,E1 -17921.525,E2 -17921.525} C_VEL
LIN {X 0,Y 276.083,Z 400.796,A -85,B 0,C 180,E1 -17923.057,E2 -17923.057} C_VEL
LIN {X 0,Y 274.425,Z 411.587,A -85,B 0,C 180,E1 -17924.838,E2 -17924.838} C_VEL
LIN {X 0,Y 272.908,Z 420.582,A -85,B 0,C 180,E1 -17926.681,E2 -17926.681} C_VEL
LIN {X 0,Y 271.526,Z 429.171,A -85,B 0,C 180,E1 -17928.877,E2 -17928.877} C_VEL
LIN {X 0,Y 270.242,Z 436.777,A -85,B 0,C 180,E1 -17931.351,E2 -17931.351} C_VEL
LIN {X 0,Y 269.271,Z 443.109,A -85,B 0,C 180,E1 -17934.034,E2 -17934.034} C_VEL
LIN {X 0,Y 268.784,Z 447.25,A -85,B 0,C 180,E1 -17936.391,E2 -17936.391} C_VEL
LIN {X 0,Y 268.458,Z 449.553,A -85,B 0,C 180,E1 -17938.113,E2 -17938.113} C_VEL
LIN {X 0,Y 268.053,Z 451.506,A -85,B 0,C 180,E1 -17940.116,E2 -17940.116} C_VEL
LIN {X 0,Y 267.903,Z 453.025,A -85,B 0,C 180,E1 -17942.937,E2 -17942.937} C_VEL
LIN {X 0,Y 268.062,Z 453.152,A -85,B 0,C 180,E1 -17945.654,E2 -17945.654} C_VEL
LIN {X 0,Y 268.462,Z 452.014,A -85,B 0,C 180,E1 -17948.264,E2 -17948.264} C_VEL
LIN {X 0,Y 269.164,Z 449.734,A -85,B 0,C 180,E1 -17950.799,E2 -17950.799} C_VEL
LIN {X 0,Y 270.047,Z 446.383,A -85,B 0,C 180,E1 -17953.238,E2 -17953.238} C_VEL
LIN {X 0,Y 271.244,Z 441.878,A -85,B 0,C 180,E1 -17955.622,E2 -17955.622} C_VEL
LIN {X 0,Y 272.787,Z 436.11,A -85,B 0,C 180,E1 -17957.958,E2 -17957.958} C_VEL
LIN {X 0,Y 274.681,Z 428.861,A -85,B 0,C 180,E1 -17960.248,E2 -17960.248} C_VEL
LIN {X 0,Y 276.886,Z 419.837,A -85,B 0,C 180,E1 -17962.483,E2 -17962.483} C_VEL
LIN {X 0,Y 278.965,Z 410.818,A -85,B 0,C 180,E1 -17964.265,E2 -17964.265} C_VEL
LIN {X 0,Y 281.044,Z 400.552,A -85,B 0,C 180,E1 -17965.89,E2 -17965.89} C_VEL
LIN {X 0,Y 283.03,Z 389.419,A -85,B 0,C 180,E1 -17967.285,E2 -17967.285} C_VEL
LIN {X 0,Y 284.693,Z 378.142,A -85,B 0,C 180,E1 -17968.392,E2 -17968.392} C_VEL
LIN {X 0,Y 286.136,Z 365.493,A -85,B 0,C 180,E1 -17969.319,E2 -17969.319} C_VEL
LIN {X 0,Y 287.228,Z 351.913,A -85,B 0,C 180,E1 -17969.989,E2 -17969.989} C_VEL
LIN {X 0,Y 288.747,Z 316.449,A -85,B 0,C 180,E1 -17970.981,E2 -17970.981} C_VEL
LIN {X 0,Y 290.117,Z 281.774,A -85,B 0,C 180,E1 -17971.915,E2 -17971.915} C_VEL
LIN {X 0,Y 284.126,Z 267.882,A -85,B 0,C 180,E1 -17973.207,E2 -17973.207} C_VEL
LIN {X 0,Y 278.926,Z 257.531,A -85,B 0,C 180,E1 -17974.353,E2 -17974.353} C_VEL
LIN {X 0,Y 273.025,Z 247.119,A -85,B 0,C 180,E1 -17975.689,E2 -17975.689} C_VEL
LIN {X 0,Y 270.989,Z 243.441,A -85,B 0,C 180,E1 -17976.207,E2 -17976.207} C_VEL
LIN {X 0,Y 270.227,Z 240.825,A -85,B 0,C 180,E1 -17977.453,E2 -17977.453} C_VEL
LIN {X 0,Y 270.2,Z 240.828,A -85,B 0,C 180,E1 -17978.223,E2 -17978.223} C_VEL
LIN {X 0,Y 269.547,Z 240.915,A -85,B 0,C 180,E1 -17979.467,E2 -17979.467} C_VEL
LIN {X 0,Y 266.796,Z 241.26,A -85,B 0,C 180,E1 -17981.497,E2 -17981.497} C_VEL
LIN {X 0,Y 263.643,Z 241.648,A -85,B 0,C 180,E1 -17983.993,E2 -17983.993} C_VEL
LIN {X 0,Y 263.302,Z 241.685,A -85,B 0,C 180,E1 -17984.855,E2 -17984.855} C_VEL
LIN {X 0,Y 263.34,Z 241.681,A -85,B 0,C 180,E1 -17989.242,E2 -17989.242} C_VEL
LIN {X 0,Y 263.526,Z 241.656,A -85,B 0,C 180,E1 -17992.346,E2 -17992.346} C_VEL
LIN {X 0,Y 263.739,Z 241.624,A -85,B 0,C 180,E1 -17998.482,E2 -17998.482} C_VEL
LIN {X 0,Y 263.733,Z 241.625,A -85,B 0,C 180,E1 -18001.536,E2 -18001.536} C_VEL
LIN {X 0,Y 263.533,Z 241.656,A -85,B 0,C 180,E1 -18007.671,E2 -18007.671} C_VEL
LIN {X 0,Y 263.348,Z 241.672,A -85,B 0,C 180,E1 -18010.775,E2 -18010.775} C_VEL
LIN {X 0,Y 263.312,Z 241.682,A -85,B 0,C 180,E1 -18015.488,E2 -18015.488} C_VEL
LIN {X 0,Y 263.213,Z 241.697,A -85,B 0,C 180,E1 -18020.319,E2 -18020.319} C_VEL
LIN {X 0,Y 263.127,Z 241.705,A -85,B 0,C 180,E1 -18025.308,E2 -18025.308} C_VEL
LIN {X 0,Y 263.126,Z 241.707,A -85,B 0,C 180,E1 -18028.744,E2 -18028.744} C_VEL
LIN {X 0,Y 263.128,Z 241.708,A -85,B 0,C 180,E1 -18032.297,E2 -18032.297} C_VEL
LIN {X 0,Y 263.163,Z 241.702,A -85,B 0,C 180,E1 -18035.99,E2 -18035.99} C_VEL
LIN {X 0,Y 263.081,Z 241.711,A -85,B 0,C 180,E1 -18039.885,E2 -18039.885} C_VEL
LIN {X 0,Y 263.08,Z 241.721,A -85,B 0,C 180,E1 -18044.002,E2 -18044.002} C_VEL
LIN {X 0,Y 263.075,Z 241.721,A -85,B 0,C 180,E1 -18048.428,E2 -18048.428} C_VEL
LIN {X 0,Y 263.112,Z 241.83,A -85,B 0,C 180,E1 -18049.271,E2 -18049.271} C_VEL
LIN {X 0,Y 265.644,Z 250.244,A -85,B 0,C 180,E1 -18053.094,E2 -18053.094} C_VEL
LIN {X 0,Y 267.57,Z 258.053,A -85,B 0,C 180,E1 -18056.263,E2 -18056.263} C_VEL
LIN {X 0,Y 274.304,Z 271.585,A -85,B 0,C 180,E1 -18057.908,E2 -18057.908} C_VEL
LIN {X 0,Y 279.238,Z 283.217,A -85,B 0,C 180,E1 -18059.086,E2 -18059.086} C_VEL
LIN {X 0,Y 282.385,Z 303.354,A -85,B 0,C 180,E1 -18060.231,E2 -18060.231} C_VEL
LIN {X 0,Y 283.179,Z 310.927,A -85,B 0,C 180,E1 -18060.591,E2 -18060.591} C_VEL
LIN {X 0,Y 280.73,Z 368.595,A -85,B 0,C 180,E1 -18062.208,E2 -18062.208} C_VEL
LIN {X 0,Y 279.367,Z 382.553,A -85,B 0,C 180,E1 -18062.874,E2 -18062.874} C_VEL
LIN {X 0,Y 277.761,Z 394.526,A -85,B 0,C 180,E1 -18063.719,E2 -18063.719} C_VEL
LIN {X 0,Y 275.557,Z 407.001,A -85,B 0,C 180,E1 -18064.912,E2 -18064.912} C_VEL
LIN {X 0,Y 273.4,Z 418.176,A -85,B 0,C 180,E1 -18066.319,E2 -18066.319} C_VEL
LIN {X 0,Y 271.088,Z 428.323,A -85,B 0,C 180,E1 -18067.92,E2 -18067.92} C_VEL
LIN {X 0,Y 268.85,Z 437.494,A -85,B 0,C 180,E1 -18069.735,E2 -18069.735} C_VEL
LIN {X 0,Y 266.704,Z 446.485,A -85,B 0,C 180,E1 -18071.964,E2 -18071.964} C_VEL
LIN {X 0,Y 264.87,Z 453.76,A -85,B 0,C 180,E1 -18074.219,E2 -18074.219} C_VEL
LIN {X 0,Y 263.495,Z 458.69,A -85,B 0,C 180,E1 -18076.111,E2 -18076.111} C_VEL
LIN {X 0,Y 262.388,Z 463.505,A -85,B 0,C 180,E1 -18078.412,E2 -18078.412} C_VEL
LIN {X 0,Y 261.682,Z 467.214,A -85,B 0,C 180,E1 -18080.727,E2 -18080.727} C_VEL
LIN {X 0,Y 261.335,Z 469.145,A -85,B 0,C 180,E1 -18082.273,E2 -18082.273} C_VEL
LIN {X 0,Y 261.109,Z 471.392,A -85,B 0,C 180,E1 -18084.864,E2 -18084.864} C_VEL
LIN {X 0,Y 261.109,Z 472.346,A -85,B 0,C 180,E1 -18086.914,E2 -18086.914} C_VEL
LIN {X 0,Y 261.147,Z 472.623,A -85,B 0,C 180,E1 -18088.458,E2 -18088.458} C_VEL
LIN {X 0,Y 261.169,Z 472.458,A -85,B 0,C 180,E1 -18090,E2 -18090} C_VEL
LIN {X 0,Y 261.155,Z 471.883,A -85,B 0,C 180,E1 -18091.542,E2 -18091.542} C_VEL
LIN {X 0,Y 261.121,Z 470.905,A -85,B 0,C 180,E1 -18093.086,E2 -18093.086} C_VEL
LIN {X 0,Y 261.147,Z 468.821,A -85,B 0,C 180,E1 -18095.23,E2 -18095.23} C_VEL
LIN {X 0,Y 261.358,Z 465.308,A -85,B 0,C 180,E1 -18097.727,E2 -18097.727} C_VEL
LIN {X 0,Y 261.783,Z 460.891,A -85,B 0,C 180,E1 -18100.05,E2 -18100.05} C_VEL
LIN {X 0,Y 262.496,Z 455.243,A -85,B 0,C 180,E1 -18102.368,E2 -18102.368} C_VEL
LIN {X 0,Y 263.74,Z 448.18,A -85,B 0,C 180,E1 -18104.664,E2 -18104.664} C_VEL
LIN {X 0,Y 265.227,Z 439.294,A -85,B 0,C 180,E1 -18106.946,E2 -18106.946} C_VEL
LIN {X 0,Y 266.67,Z 430.173,A -85,B 0,C 180,E1 -18108.835,E2 -18108.835} C_VEL
LIN {X 0,Y 268.232,Z 420.131,A -85,B 0,C 180,E1 -18110.514,E2 -18110.514} C_VEL
LIN {X 0,Y 269.908,Z 408.989,A -85,B 0,C 180,E1 -18111.981,E2 -18111.981} C_VEL
LIN {X 0,Y 271.545,Z 396.543,A -85,B 0,C 180,E1 -18113.246,E2 -18113.246} C_VEL
LIN {X 0,Y 272.813,Z 384.747,A -85,B 0,C 180,E1 -18114.139,E2 -18114.139} C_VEL
LIN {X 0,Y 273.792,Z 372.054,A -85,B 0,C 180,E1 -18114.804,E2 -18114.804} C_VEL
LIN {X 0,Y 274.47,Z 354.823,A -85,B 0,C 180,E1 -18115.346,E2 -18115.346} C_VEL
LIN {X 0,Y 275.849,Z 307.716,A -85,B 0,C 180,E1 -18116.641,E2 -18116.641} C_VEL
LIN {X 0,Y 270.683,Z 270.673,A -85,B 0,C 180,E1 -18118.23,E2 -18118.23} C_VEL
LIN {X 0,Y 267.102,Z 260.345,A -85,B 0,C 180,E1 -18118.91,E2 -18118.91} C_VEL
LIN {X 0,Y 265.031,Z 250.1,A -85,B 0,C 180,E1 -18122.477,E2 -18122.477} C_VEL
LIN {X 0,Y 263.206,Z 241.699,A -85,B 0,C 180,E1 -18125.581,E2 -18125.581} C_VEL
LIN {X 0,Y 263.083,Z 241.718,A -85,B 0,C 180,E1 -18129.875,E2 -18129.875} C_VEL
LIN {X 0,Y 263.068,Z 241.72,A -85,B 0,C 180,E1 -18133.994,E2 -18133.994} C_VEL
LIN {X 0,Y 263.072,Z 241.714,A -85,B 0,C 180,E1 -18138.418,E2 -18138.418} C_VEL
LIN {X 0,Y 263.116,Z 241.711,A -85,B 0,C 180,E1 -18142.087,E2 -18142.087} C_VEL
LIN {X 0,Y 263.164,Z 241.707,A -85,B 0,C 180,E1 -18145.879,E2 -18145.879} C_VEL
LIN {X 0,Y 263.118,Z 241.71,A -85,B 0,C 180,E1 -18149.495,E2 -18149.495} C_VEL
LIN {X 0,Y 263.12,Z 241.707,A -85,B 0,C 180,E1 -18152.987,E2 -18152.987} C_VEL
LIN {X 0,Y 263.123,Z 241.707,A -85,B 0,C 180,E1 -18156.373,E2 -18156.373} C_VEL
LIN {X 0,Y 263.213,Z 241.691,A -85,B 0,C 180,E1 -18159.681,E2 -18159.681} C_VEL
LIN {X 0,Y 263.312,Z 241.676,A -85,B 0,C 180,E1 -18164.512,E2 -18164.512} C_VEL
LIN {X 0,Y 263.332,Z 241.683,A -85,B 0,C 180,E1 -18169.225,E2 -18169.225} C_VEL
LIN {X 0,Y 263.511,Z 241.653,A -85,B 0,C 180,E1 -18172.328,E2 -18172.328} C_VEL
LIN {X 0,Y 263.721,Z 241.618,A -85,B 0,C 180,E1 -18178.464,E2 -18178.464} C_VEL
LIN {X 0,Y 263.725,Z 241.63,A -85,B 0,C 180,E1 -18181.518,E2 -18181.518} C_VEL
LIN {X 0,Y 263.512,Z 241.658,A -85,B 0,C 180,E1 -18187.654,E2 -18187.654} C_VEL
LIN {X 0,Y 263.334,Z 241.677,A -85,B 0,C 180,E1 -18190.758,E2 -18190.758} C_VEL
LIN {X 0,Y 263.305,Z 241.686,A -85,B 0,C 180,E1 -18195.471,E2 -18195.471} C_VEL
LIN {X 0,Y 263.24,Z 241.689,A -85,B 0,C 180,E1 -18200.298,E2 -18200.298} C_VEL
LIN {X 0,Y 263.16,Z 241.704,A -85,B 0,C 180,E1 -18205.285,E2 -18205.285} C_VEL
LIN {X 0,Y 263.125,Z 241.697,A -85,B 0,C 180,E1 -18208.724,E2 -18208.724} C_VEL
LIN {X 0,Y 263.097,Z 241.69,A -85,B 0,C 180,E1 -18212.281,E2 -18212.281} C_VEL
LIN {X 0,Y 263.143,Z 241.701,A -85,B 0,C 180,E1 -18216.753,E2 -18216.753} C_VEL
LIN {X 0,Y 263.069,Z 241.714,A -85,B 0,C 180,E1 -18219.865,E2 -18219.865} C_VEL
LIN {X 0,Y 263.086,Z 241.709,A -85,B 0,C 180,E1 -18223.977,E2 -18223.977} C_VEL
LIN {X 0,Y 263.083,Z 241.712,A -85,B 0,C 180,E1 -18228.4,E2 -18228.4} C_VEL
LIN {X 0,Y 263.137,Z 241.71,A -85,B 0,C 180,E1 -18233.231,E2 -18233.231} C_VEL
LIN {X 0,Y 263.085,Z 241.714,A -85,B 0,C 180,E1 -18237.706,E2 -18237.706} C_VEL
LIN {X 0,Y 263.153,Z 241.703,A -85,B 0,C 180,E1 -18241.778,E2 -18241.778} C_VEL
LIN {X 0,Y 263.187,Z 241.706,A -85,B 0,C 180,E1 -18245.191,E2 -18245.191} C_VEL
LIN {X 0,Y 263.238,Z 241.697,A -85,B 0,C 180,E1 -18249.692,E2 -18249.692} C_VEL
LIN {X 0,Y 263.291,Z 241.689,A -85,B 0,C 180,E1 -18254.519,E2 -18254.519} C_VEL
LIN {X 0,Y 263.319,Z 241.685,A -85,B 0,C 180,E1 -18259.232,E2 -18259.232} C_VEL
LIN {X 0,Y 263.518,Z 241.658,A -85,B 0,C 180,E1 -18262.337,E2 -18262.337} C_VEL
LIN {X 0,Y 263.702,Z 241.637,A -85,B 0,C 180,E1 -18268.473,E2 -18268.473} C_VEL
LIN {X 0,Y 263.702,Z 241.636,A -85,B 0,C 180,E1 -18271.527,E2 -18271.527} C_VEL
LIN {X 0,Y 263.469,Z 241.772,A -85,B 0,C 180,E1 -18273.584,E2 -18273.584} C_VEL
LIN {X 0,Y 263.608,Z 242.669,A -85,B 0,C 180,E1 -18273.845,E2 -18273.845} C_VEL
LIN {X 0,Y 271.621,Z 262.559,A -85,B 0,C 180,E1 -18275.249,E2 -18275.249} C_VEL
LIN {X 0,Y 276.744,Z 277.398,A -85,B 0,C 180,E1 -18276.159,E2 -18276.159} C_VEL
LIN {X 0,Y 274.365,Z 349.396,A -85,B 0,C 180,E1 -18278.145,E2 -18278.145} C_VEL
LIN {X 0,Y 273.443,Z 362.622,A -85,B 0,C 180,E1 -18278.778,E2 -18278.778} C_VEL
LIN {X 0,Y 272.375,Z 375.995,A -85,B 0,C 180,E1 -18279.749,E2 -18279.749} C_VEL
LIN {X 0,Y 271.167,Z 387.006,A -85,B 0,C 180,E1 -18280.829,E2 -18280.829} C_VEL
LIN {X 0,Y 269.688,Z 398.115,A -85,B 0,C 180,E1 -18282.224,E2 -18282.224} C_VEL
LIN {X 0,Y 267.954,Z 409.404,A -85,B 0,C 180,E1 -18284.012,E2 -18284.012} C_VEL
LIN {X 0,Y 266.496,Z 417.877,A -85,B 0,C 180,E1 -18285.682,E2 -18285.682} C_VEL
LIN {X 0,Y 264.927,Z 427.177,A -85,B 0,C 180,E1 -18287.97,E2 -18287.97} C_VEL
LIN {X 0,Y 263.665,Z 434.642,A -85,B 0,C 180,E1 -18290.274,E2 -18290.274} C_VEL
LIN {X 0,Y 262.595,Z 441.132,A -85,B 0,C 180,E1 -18292.834,E2 -18292.834} C_VEL
LIN {X 0,Y 261.843,Z 446.121,A -85,B 0,C 180,E1 -18295.432,E2 -18295.432} C_VEL
LIN {X 0,Y 261.505,Z 449.163,A -85,B 0,C 180,E1 -18297.542,E2 -18297.542} C_VEL
LIN {X 0,Y 260.911,Z 452.026,A -85,B 0,C 180,E1 -18300.485,E2 -18300.485} C_VEL
LIN {X 0,Y 260.825,Z 453.384,A -85,B 0,C 180,E1 -18303.374,E2 -18303.374} C_VEL
LIN {X 0,Y 261.032,Z 453.285,A -85,B 0,C 180,E1 -18306.321,E2 -18306.321} C_VEL
LIN {X 0,Y 261.499,Z 452.081,A -85,B 0,C 180,E1 -18308.813,E2 -18308.813} C_VEL
LIN {X 0,Y 262.284,Z 449.69,A -85,B 0,C 180,E1 -18311.403,E2 -18311.403} C_VEL
LIN {X 0,Y 263.307,Z 446.149,A -85,B 0,C 180,E1 -18313.944,E2 -18313.944} C_VEL
LIN {X 0,Y 264.578,Z 441.6,A -85,B 0,C 180,E1 -18316.334,E2 -18316.334} C_VEL
LIN {X 0,Y 266.224,Z 435.697,A -85,B 0,C 180,E1 -18318.717,E2 -18318.717} C_VEL
LIN {X 0,Y 268.292,Z 428.218,A -85,B 0,C 180,E1 -18321.06,E2 -18321.06} C_VEL
LIN {X 0,Y 270.69,Z 418.993,A -85,B 0,C 180,E1 -18323.347,E2 -18323.347} C_VEL
LIN {X 0,Y 272.892,Z 409.651,A -85,B 0,C 180,E1 -18325.173,E2 -18325.173} C_VEL
LIN {X 0,Y 275.06,Z 399.225,A -85,B 0,C 180,E1 -18326.805,E2 -18326.805} C_VEL
LIN {X 0,Y 277.081,Z 388.372,A -85,B 0,C 180,E1 -18328.147,E2 -18328.147} C_VEL
LIN {X 0,Y 278.778,Z 377.158,A -85,B 0,C 180,E1 -18329.233,E2 -18329.233} C_VEL
LIN {X 0,Y 280.258,Z 364.171,A -85,B 0,C 180,E1 -18330.16,E2 -18330.16} C_VEL
LIN {X 0,Y 281.272,Z 351.398,A -85,B 0,C 180,E1 -18330.782,E2 -18330.782} C_VEL
LIN {X 0,Y 284.163,Z 283.642,A -85,B 0,C 180,E1 -18332.671,E2 -18332.671} C_VEL
LIN {X 0,Y 277.645,Z 268.624,A -85,B 0,C 180,E1 -18334.164,E2 -18334.164} C_VEL
LIN {X 0,Y 270.445,Z 255.126,A -85,B 0,C 180,E1 -18335.835,E2 -18335.835} C_VEL
LIN {X 0,Y 265.67,Z 247.23,A -85,B 0,C 180,E1 -18336.993,E2 -18336.993} C_VEL
LIN {X 0,Y 263.816,Z 243.846,A -85,B 0,C 180,E1 -18337.494,E2 -18337.494} C_VEL
LIN {X 0,Y 263.173,Z 241.705,A -85,B 0,C 180,E1 -18338.584,E2 -18338.584} C_VEL
LIN {X 0,Y 263.25,Z 241.692,A -85,B 0,C 180,E1 -18342.932,E2 -18342.932} C_VEL
LIN {X 0,Y 263.302,Z 241.685,A -85,B 0,C 180,E1 -18344.855,E2 -18344.855} C_VEL
LIN {X 0,Y 262.594,Z 241.776,A -85,B 0,C 180,E1 -18346.131,E2 -18346.131} C_VEL
LIN {X 0,Y 259.774,Z 242.121,A -85,B 0,C 180,E1 -18348.215,E2 -18348.215} C_VEL
LIN {X 0,Y 257.446,Z 242.418,A -85,B 0,C 180,E1 -18349.909,E2 -18349.909} C_VEL
LIN {X 0,Y 256.499,Z 242.528,A -85,B 0,C 180,E1 -18351.221,E2 -18351.221} C_VEL
LIN {X 0,Y 256.447,Z 242.534,A -85,B 0,C 180,E1 -18351.664,E2 -18351.664} C_VEL
LIN {X 0,Y 256.456,Z 242.538,A -85,B 0,C 180,E1 -18353.716,E2 -18353.716} C_VEL
LIN {X 0,Y 256.703,Z 242.5,A -85,B 0,C 180,E1 -18358.44,E2 -18358.44} C_VEL
LIN {X 0,Y 256.695,Z 242.501,A -85,B 0,C 180,E1 -18361.578,E2 -18361.578} C_VEL
LIN {X 0,Y 256.459,Z 242.528,A -85,B 0,C 180,E1 -18366.302,E2 -18366.302} C_VEL
LIN {X 0,Y 256.426,Z 242.534,A -85,B 0,C 180,E1 -18369.473,E2 -18369.473} C_VEL
LIN {X 0,Y 256.232,Z 242.557,A -85,B 0,C 180,E1 -18374.3,E2 -18374.3} C_VEL
LIN {X 0,Y 256.159,Z 242.571,A -85,B 0,C 180,E1 -18377.574,E2 -18377.574} C_VEL
LIN {X 0,Y 256.124,Z 242.578,A -85,B 0,C 180,E1 -18381.104,E2 -18381.104} C_VEL
LIN {X 0,Y 256.089,Z 242.582,A -85,B 0,C 180,E1 -18385.094,E2 -18385.094} C_VEL
LIN {X 0,Y 256.085,Z 242.585,A -85,B 0,C 180,E1 -18388.576,E2 -18388.576} C_VEL
LIN {X 0,Y 256.074,Z 242.587,A -85,B 0,C 180,E1 -18391.704,E2 -18391.704} C_VEL
LIN {X 0,Y 256.089,Z 242.586,A -85,B 0,C 180,E1 -18395.2,E2 -18395.2} C_VEL
LIN {X 0,Y 256.054,Z 242.587,A -85,B 0,C 180,E1 -18399.154,E2 -18399.154} C_VEL
LIN {X 0,Y 256.004,Z 242.6,A -85,B 0,C 180,E1 -18403.348,E2 -18403.348} C_VEL
LIN {X 0,Y 256.005,Z 242.6,A -85,B 0,C 180,E1 -18406.663,E2 -18406.663} C_VEL
LIN {X 0,Y 256.066,Z 242.725,A -85,B 0,C 180,E1 -18408.038,E2 -18408.038} C_VEL
LIN {X 0,Y 258.591,Z 251.006,A -85,B 0,C 180,E1 -18412.024,E2 -18412.024} C_VEL
LIN {X 0,Y 260.294,Z 257.596,A -85,B 0,C 180,E1 -18414.884,E2 -18414.884} C_VEL
LIN {X 0,Y 262.604,Z 262.074,A -85,B 0,C 180,E1 -18415.51,E2 -18415.51} C_VEL
LIN {X 0,Y 268.133,Z 272.998,A -85,B 0,C 180,E1 -18416.928,E2 -18416.928} C_VEL
LIN {X 0,Y 273.726,Z 285.764,A -85,B 0,C 180,E1 -18418.322,E2 -18418.322} C_VEL
LIN {X 0,Y 276.68,Z 305.362,A -85,B 0,C 180,E1 -18419.469,E2 -18419.469} C_VEL
LIN {X 0,Y 277.33,Z 311.292,A -85,B 0,C 180,E1 -18419.771,E2 -18419.771} C_VEL
LIN {X 0,Y 274.799,Z 368.066,A -85,B 0,C 180,E1 -18421.398,E2 -18421.398} C_VEL
LIN {X 0,Y 273.394,Z 382.093,A -85,B 0,C 180,E1 -18422.074,E2 -18422.074} C_VEL
LIN {X 0,Y 271.635,Z 394.62,A -85,B 0,C 180,E1 -18422.975,E2 -18422.975} C_VEL
LIN {X 0,Y 269.526,Z 406.232,A -85,B 0,C 180,E1 -18424.103,E2 -18424.103} C_VEL
LIN {X 0,Y 267.213,Z 417.502,A -85,B 0,C 180,E1 -18425.529,E2 -18425.529} C_VEL
LIN {X 0,Y 264.801,Z 427.735,A -85,B 0,C 180,E1 -18427.161,E2 -18427.161} C_VEL
LIN {X 0,Y 262.22,Z 437.786,A -85,B 0,C 180,E1 -18429.2,E2 -18429.2} C_VEL
LIN {X 0,Y 259.971,Z 446.664,A -85,B 0,C 180,E1 -18431.48,E2 -18431.48} C_VEL
LIN {X 0,Y 258.046,Z 453.826,A -85,B 0,C 180,E1 -18433.79,E2 -18433.79} C_VEL
LIN {X 0,Y 256.147,Z 460.398,A -85,B 0,C 180,E1 -18436.514,E2 -18436.514} C_VEL
LIN {X 0,Y 255.105,Z 464.776,A -85,B 0,C 180,E1 -18438.881,E2 -18438.881} C_VEL
LIN {X 0,Y 254.637,Z 467.111,A -85,B 0,C 180,E1 -18440.468,E2 -18440.468} C_VEL
LIN {X 0,Y 254.277,Z 469.001,A -85,B 0,C 180,E1 -18442.057,E2 -18442.057} C_VEL
LIN {X 0,Y 253.998,Z 471.471,A -85,B 0,C 180,E1 -18445.239,E2 -18445.239} C_VEL
LIN {X 0,Y 254.004,Z 472.118,A -85,B 0,C 180,E1 -18446.828,E2 -18446.828} C_VEL
LIN {X 0,Y 254.075,Z 472.357,A -85,B 0,C 180,E1 -18448.415,E2 -18448.415} C_VEL
LIN {X 0,Y 254.096,Z 472.156,A -85,B 0,C 180,E1 -18450,E2 -18450} C_VEL
LIN {X 0,Y 254.083,Z 471.557,A -85,B 0,C 180,E1 -18451.585,E2 -18451.585} C_VEL
LIN {X 0,Y 254.036,Z 470.555,A -85,B 0,C 180,E1 -18453.172,E2 -18453.172} C_VEL
LIN {X 0,Y 254.045,Z 468.711,A -85,B 0,C 180,E1 -18455.118,E2 -18455.118} C_VEL
LIN {X 0,Y 254.312,Z 464.853,A -85,B 0,C 180,E1 -18457.942,E2 -18457.942} C_VEL
LIN {X 0,Y 254.756,Z 460.376,A -85,B 0,C 180,E1 -18460.33,E2 -18460.33} C_VEL
LIN {X 0,Y 255.526,Z 454.663,A -85,B 0,C 180,E1 -18462.711,E2 -18462.711} C_VEL
LIN {X 0,Y 256.822,Z 447.491,A -85,B 0,C 180,E1 -18465.068,E2 -18465.068} C_VEL
LIN {X 0,Y 258.376,Z 438.51,A -85,B 0,C 180,E1 -18467.41,E2 -18467.41} C_VEL
LIN {X 0,Y 259.908,Z 429.283,A -85,B 0,C 180,E1 -18469.344,E2 -18469.344} C_VEL
LIN {X 0,Y 261.514,Z 419.04,A -85,B 0,C 180,E1 -18471.066,E2 -18471.066} C_VEL
LIN {X 0,Y 263.27,Z 407.702,A -85,B 0,C 180,E1 -18472.565,E2 -18472.565} C_VEL
LIN {X 0,Y 264.88,Z 396,A -85,B 0,C 180,E1 -18473.763,E2 -18473.763} C_VEL
LIN {X 0,Y 266.155,Z 384.065,A -85,B 0,C 180,E1 -18474.679,E2 -18474.679} C_VEL
LIN {X 0,Y 267.211,Z 371.187,A -85,B 0,C 180,E1 -18475.354,E2 -18475.354} C_VEL
LIN {X 0,Y 268.019,Z 350.346,A -85,B 0,C 180,E1 -18476.001,E2 -18476.001} C_VEL
LIN {X 0,Y 269.274,Z 308.822,A -85,B 0,C 180,E1 -18477.171,E2 -18477.171} C_VEL
LIN {X 0,Y 264.598,Z 274.519,A -85,B 0,C 180,E1 -18478.678,E2 -18478.678} C_VEL
LIN {X 0,Y 263.713,Z 270.851,A -85,B 0,C 180,E1 -18478.881,E2 -18478.881} C_VEL
LIN {X 0,Y 259.833,Z 259.998,A -85,B 0,C 180,E1 -18479.66,E2 -18479.66} C_VEL
LIN {X 0,Y 257.642,Z 249.288,A -85,B 0,C 180,E1 -18483.53,E2 -18483.53} C_VEL
LIN {X 0,Y 256.139,Z 242.577,A -85,B 0,C 180,E1 -18486.15,E2 -18486.15} C_VEL
LIN {X 0,Y 256.04,Z 242.594,A -85,B 0,C 180,E1 -18489.765,E2 -18489.765} C_VEL
LIN {X 0,Y 256.013,Z 242.597,A -85,B 0,C 180,E1 -18494.45,E2 -18494.45} C_VEL
LIN {X 0,Y 256.011,Z 242.594,A -85,B 0,C 180,E1 -18498.779,E2 -18498.779} C_VEL
LIN {X 0,Y 256.113,Z 242.581,A -85,B 0,C 180,E1 -18502.856,E2 -18502.856} C_VEL
LIN {X 0,Y 256.074,Z 242.587,A -85,B 0,C 180,E1 -18506.7,E2 -18506.7} C_VEL
LIN {X 0,Y 256.05,Z 242.59,A -85,B 0,C 180,E1 -18510.384,E2 -18510.384} C_VEL
LIN {X 0,Y 256.074,Z 242.587,A -85,B 0,C 180,E1 -18513.944,E2 -18513.944} C_VEL
LIN {X 0,Y 256.064,Z 242.589,A -85,B 0,C 180,E1 -18517.395,E2 -18517.395} C_VEL
LIN {X 0,Y 256.113,Z 242.57,A -85,B 0,C 180,E1 -18520.766,E2 -18520.766} C_VEL
LIN {X 0,Y 256.232,Z 242.559,A -85,B 0,C 180,E1 -18524.072,E2 -18524.072} C_VEL
LIN {X 0,Y 256.278,Z 242.56,A -85,B 0,C 180,E1 -18528.924,E2 -18528.924} C_VEL
LIN {X 0,Y 256.453,Z 242.533,A -85,B 0,C 180,E1 -18532.116,E2 -18532.116} C_VEL
LIN {X 0,Y 256.281,Z 242.541,A -85,B 0,C 180,E1 -18535.272,E2 -18535.272} C_VEL
LIN {X 0,Y 256.682,Z 242.494,A -85,B 0,C 180,E1 -18538.422,E2 -18538.422} C_VEL
LIN {X 0,Y 256.687,Z 242.506,A -85,B 0,C 180,E1 -18541.56,E2 -18541.56} C_VEL
LIN {X 0,Y 256.429,Z 242.538,A -85,B 0,C 180,E1 -18546.559,E2 -18546.559} C_VEL
LIN {X 0,Y 256.414,Z 242.539,A -85,B 0,C 180,E1 -18549.456,E2 -18549.456} C_VEL
LIN {X 0,Y 256.219,Z 242.567,A -85,B 0,C 180,E1 -18554.282,E2 -18554.282} C_VEL
LIN {X 0,Y 256.164,Z 242.57,A -85,B 0,C 180,E1 -18557.555,E2 -18557.555} C_VEL
LIN {X 0,Y 256.132,Z 242.577,A -85,B 0,C 180,E1 -18561.108,E2 -18561.108} C_VEL
LIN {X 0,Y 256.141,Z 242.578,A -85,B 0,C 180,E1 -18565.119,E2 -18565.119} C_VEL
LIN {X 0,Y 256.085,Z 242.572,A -85,B 0,C 180,E1 -18568.576,E2 -18568.576} C_VEL
LIN {X 0,Y 256.043,Z 242.566,A -85,B 0,C 180,E1 -18571.692,E2 -18571.692} C_VEL
LIN {X 0,Y 256.047,Z 242.58,A -85,B 0,C 180,E1 -18575.185,E2 -18575.185} C_VEL
LIN {X 0,Y 256.076,Z 242.584,A -85,B 0,C 180,E1 -18577.261,E2 -18577.261} C_VEL
LIN {X 0,Y 256.018,Z 242.595,A -85,B 0,C 180,E1 -18581.196,E2 -18581.196} C_VEL
LIN {X 0,Y 256.021,Z 242.594,A -85,B 0,C 180,E1 -18585.522,E2 -18585.522} C_VEL
LIN {X 0,Y 256.013,Z 242.594,A -85,B 0,C 180,E1 -18588.79,E2 -18588.79} C_VEL
LIN {X 0,Y 256.086,Z 242.585,A -85,B 0,C 180,E1 -18592.861,E2 -18592.861} C_VEL
LIN {X 0,Y 256.022,Z 242.591,A -85,B 0,C 180,E1 -18596.701,E2 -18596.701} C_VEL
LIN {X 0,Y 256.066,Z 242.588,A -85,B 0,C 180,E1 -18600.395,E2 -18600.395} C_VEL
LIN {X 0,Y 256.147,Z 242.581,A -85,B 0,C 180,E1 -18604.853,E2 -18604.853} C_VEL
LIN {X 0,Y 256.188,Z 242.577,A -85,B 0,C 180,E1 -18609.107,E2 -18609.107} C_VEL
LIN {X 0,Y 256.241,Z 242.567,A -85,B 0,C 180,E1 -18614.082,E2 -18614.082} C_VEL
LIN {X 0,Y 256.255,Z 242.566,A -85,B 0,C 180,E1 -18618.932,E2 -18618.932} C_VEL
LIN {X 0,Y 256.486,Z 242.533,A -85,B 0,C 180,E1 -18622.126,E2 -18622.126} C_VEL
LIN {X 0,Y 256.666,Z 242.514,A -85,B 0,C 180,E1 -18628.431,E2 -18628.431} C_VEL
LIN {X 0,Y 256.667,Z 242.512,A -85,B 0,C 180,E1 -18631.569,E2 -18631.569} C_VEL
LIN {X 0,Y 256.532,Z 242.631,A -85,B 0,C 180,E1 -18633.092,E2 -18633.092} C_VEL
LIN {X 0,Y 258.56,Z 248.183,A -85,B 0,C 180,E1 -18633.507,E2 -18633.507} C_VEL
LIN {X 0,Y 265.003,Z 263.942,A -85,B 0,C 180,E1 -18634.667,E2 -18634.667} C_VEL
LIN {X 0,Y 270.133,Z 278.713,A -85,B 0,C 180,E1 -18635.612,E2 -18635.612} C_VEL
LIN {X 0,Y 267.712,Z 350.043,A -85,B 0,C 180,E1 -18637.637,E2 -18637.637} C_VEL
LIN {X 0,Y 266.722,Z 363.91,A -85,B 0,C 180,E1 -18638.332,E2 -18638.332} C_VEL
LIN {X 0,Y 265.63,Z 376.83,A -85,B 0,C 180,E1 -18639.315,E2 -18639.315} C_VEL
LIN {X 0,Y 264.248,Z 388.474,A -85,B 0,C 180,E1 -18640.509,E2 -18640.509} C_VEL
LIN {X 0,Y 262.724,Z 399.541,A -85,B 0,C 180,E1 -18641.965,E2 -18641.965} C_VEL
LIN {X 0,Y 261.09,Z 409.642,A -85,B 0,C 180,E1 -18643.622,E2 -18643.622} C_VEL
LIN {X 0,Y 259.606,Z 417.981,A -85,B 0,C 180,E1 -18645.304,E2 -18645.304} C_VEL
LIN {X 0,Y 258.002,Z 427.138,A -85,B 0,C 180,E1 -18647.6,E2 -18647.6} C_VEL
LIN {X 0,Y 256.668,Z 434.802,A -85,B 0,C 180,E1 -18650.015,E2 -18650.015} C_VEL
LIN {X 0,Y 255.552,Z 441.323,A -85,B 0,C 180,E1 -18652.644,E2 -18652.644} C_VEL
LIN {X 0,Y 254.783,Z 446.344,A -85,B 0,C 180,E1 -18655.323,E2 -18655.323} C_VEL
LIN {X 0,Y 254.287,Z 450.018,A -85,B 0,C 180,E1 -18658.023,E2 -18658.023} C_VEL
LIN {X 0,Y 253.798,Z 452.539,A -85,B 0,C 180,E1 -18660.882,E2 -18660.882} C_VEL
LIN {X 0,Y 253.732,Z 453.693,A -85,B 0,C 180,E1 -18663.824,E2 -18663.824} C_VEL
LIN {X 0,Y 253.979,Z 453.522,A -85,B 0,C 180,E1 -18666.652,E2 -18666.652} C_VEL
LIN {X 0,Y 254.56,Z 452.131,A -85,B 0,C 180,E1 -18669.418,E2 -18669.418} C_VEL
LIN {X 0,Y 255.408,Z 449.657,A -85,B 0,C 180,E1 -18672.034,E2 -18672.034} C_VEL
LIN {X 0,Y 256.539,Z 446.06,A -85,B 0,C 180,E1 -18674.595,E2 -18674.595} C_VEL
LIN {X 0,Y 258.075,Z 440.761,A -85,B 0,C 180,E1 -18677.329,E2 -18677.329} C_VEL
LIN {X 0,Y 260,Z 434.286,A -85,B 0,C 180,E1 -18679.859,E2 -18679.859} C_VEL
LIN {X 0,Y 262.156,Z 426.987,A -85,B 0,C 180,E1 -18682.096,E2 -18682.096} C_VEL
LIN {X 0,Y 264.549,Z 418.13,A -85,B 0,C 180,E1 -18684.249,E2 -18684.249} C_VEL
LIN {X 0,Y 266.815,Z 408.782,A -85,B 0,C 180,E1 -18686.068,E2 -18686.068} C_VEL
LIN {X 0,Y 269.126,Z 398.175,A -85,B 0,C 180,E1 -18687.717,E2 -18687.717} C_VEL
LIN {X 0,Y 271.246,Z 386.639,A -85,B 0,C 180,E1 -18689.12,E2 -18689.12} C_VEL
LIN {X 0,Y 273.145,Z 374.143,A -85,B 0,C 180,E1 -18690.269,E2 -18690.269} C_VEL
LIN {X 0,Y 274.616,Z 360.991,A -85,B 0,C 180,E1 -18691.147,E2 -18691.147} C_VEL
LIN {X 0,Y 275.598,Z 347.197,A -85,B 0,C 180,E1 -18691.732,E2 -18691.732} C_VEL
LIN {X 0,Y 278.319,Z 285.564,A -85,B 0,C 180,E1 -18693.467,E2 -18693.467} C_VEL
LIN {X 0,Y 271.883,Z 271.014,A -85,B 0,C 180,E1 -18695,E2 -18695} C_VEL
LIN {X 0,Y 264.475,Z 257.088,A -85,B 0,C 180,E1 -18696.831,E2 -18696.831} C_VEL
LIN {X 0,Y 258.85,Z 248.124,A -85,B 0,C 180,E1 -18698.282,E2 -18698.282} C_VEL
LIN {X 0,Y 256.542,Z 244.206,A -85,B 0,C 180,E1 -18698.96,E2 -18698.96} C_VEL
LIN {X 0,Y 256.2,Z 242.572,A -85,B 0,C 180,E1 -18699.853,E2 -18699.853} C_VEL
LIN {X 0,Y 256.276,Z 242.566,A -85,B 0,C 180,E1 -18704.094,E2 -18704.094} C_VEL
LIN {X 0,Y 256.278,Z 242.562,A -85,B 0,C 180,E1 -18707.337,E2 -18707.337} C_VEL
LIN {X 0,Y 256.447,Z 242.534,A -85,B 0,C 180,E1 -18711.664,E2 -18711.664} C_VEL
LIN {X 0,Y 255.87,Z 242.614,A -85,B 0,C 180,E1 -18712.972,E2 -18712.972} C_VEL
LIN {X 0,Y 253.137,Z 242.948,A -85,B 0,C 180,E1 -18715.108,E2 -18715.108} C_VEL
LIN {X 0,Y 250.77,Z 243.248,A -85,B 0,C 180,E1 -18716.846,E2 -18716.846} C_VEL
LIN {X 0,Y 249.744,Z 243.368,A -85,B 0,C 180,E1 -18718.192,E2 -18718.192} C_VEL
LIN {X 0,Y 249.658,Z 243.377,A -85,B 0,C 180,E1 -18718.648,E2 -18718.648} C_VEL
LIN {X 0,Y 249.655,Z 243.377,A -85,B 0,C 180,E1 -18721.622,E2 -18721.622} C_VEL
LIN {X 0,Y 249.432,Z 243.403,A -85,B 0,C 180,E1 -18726.48,E2 -18726.48} C_VEL
LIN {X 0,Y 249.342,Z 243.414,A -85,B 0,C 180,E1 -18729.745,E2 -18729.745} C_VEL
LIN {X 0,Y 249.172,Z 243.437,A -85,B 0,C 180,E1 -18734.714,E2 -18734.714} C_VEL
LIN {X 0,Y 249.089,Z 243.447,A -85,B 0,C 180,E1 -18738.09,E2 -18738.09} C_VEL
LIN {X 0,Y 249.049,Z 243.457,A -85,B 0,C 180,E1 -18741.53,E2 -18741.53} C_VEL
LIN {X 0,Y 249.051,Z 243.456,A -85,B 0,C 180,E1 -18745.447,E2 -18745.447} C_VEL
LIN {X 0,Y 249.033,Z 243.461,A -85,B 0,C 180,E1 -18748.975,E2 -18748.975} C_VEL
LIN {X 0,Y 249.007,Z 243.465,A -85,B 0,C 180,E1 -18752.438,E2 -18752.438} C_VEL
LIN {X 0,Y 249.023,Z 243.461,A -85,B 0,C 180,E1 -18756.355,E2 -18756.355} C_VEL
LIN {X 0,Y 248.982,Z 243.47,A -85,B 0,C 180,E1 -18760.492,E2 -18760.492} C_VEL
LIN {X 0,Y 248.967,Z 243.475,A -85,B 0,C 180,E1 -18765.114,E2 -18765.114} C_VEL
LIN {X 0,Y 248.98,Z 243.588,A -85,B 0,C 180,E1 -18766.655,E2 -18766.655} C_VEL
LIN {X 0,Y 251.22,Z 250.807,A -85,B 0,C 180,E1 -18770.389,E2 -18770.389} C_VEL
LIN {X 0,Y 253.17,Z 257.381,A -85,B 0,C 180,E1 -18773.414,E2 -18773.414} C_VEL
LIN {X 0,Y 255.656,Z 261.981,A -85,B 0,C 180,E1 -18774.134,E2 -18774.134} C_VEL
LIN {X 0,Y 262.824,Z 275.943,A -85,B 0,C 180,E1 -18776.092,E2 -18776.092} C_VEL
LIN {X 0,Y 268.199,Z 288.385,A -85,B 0,C 180,E1 -18777.517,E2 -18777.517} C_VEL
LIN {X 0,Y 270.912,Z 306.144,A -85,B 0,C 180,E1 -18778.605,E2 -18778.605} C_VEL
LIN {X 0,Y 271.533,Z 312.567,A -85,B 0,C 180,E1 -18778.933,E2 -18778.933} C_VEL
LIN {X 0,Y 268.915,Z 367.929,A -85,B 0,C 180,E1 -18780.551,E2 -18780.551} C_VEL
LIN {X 0,Y 267.478,Z 381.851,A -85,B 0,C 180,E1 -18781.24,E2 -18781.24} C_VEL
LIN {X 0,Y 265.74,Z 393.829,A -85,B 0,C 180,E1 -18782.111,E2 -18782.111} C_VEL
LIN {X 0,Y 263.546,Z 405.518,A -85,B 0,C 180,E1 -18783.257,E2 -18783.257} C_VEL
LIN {X 0,Y 261.14,Z 416.832,A -85,B 0,C 180,E1 -18784.708,E2 -18784.708} C_VEL
LIN {X 0,Y 258.55,Z 427.138,A -85,B 0,C 180,E1 -18786.364,E2 -18786.364} C_VEL
LIN {X 0,Y 256.079,Z 436.443,A -85,B 0,C 180,E1 -18788.254,E2 -18788.254} C_VEL
LIN {X 0,Y 253.951,Z 444.274,A -85,B 0,C 180,E1 -18790.226,E2 -18790.226} C_VEL
LIN {X 0,Y 251.833,Z 451.707,A -85,B 0,C 180,E1 -18792.543,E2 -18792.543} C_VEL
LIN {X 0,Y 249.736,Z 458.747,A -85,B 0,C 180,E1 -18795.329,E2 -18795.329} C_VEL
LIN {X 0,Y 248.422,Z 463.426,A -85,B 0,C 180,E1 -18797.75,E2 -18797.75} C_VEL
LIN {X 0,Y 247.61,Z 467.015,A -85,B 0,C 180,E1 -18800.195,E2 -18800.195} C_VEL
LIN {X 0,Y 247.219,Z 468.847,A -85,B 0,C 180,E1 -18801.829,E2 -18801.829} C_VEL
LIN {X 0,Y 246.907,Z 471.268,A -85,B 0,C 180,E1 -18805.102,E2 -18805.102} C_VEL
LIN {X 0,Y 246.904,Z 471.89,A -85,B 0,C 180,E1 -18806.737,E2 -18806.737} C_VEL
LIN {X 0,Y 246.98,Z 472.08,A -85,B 0,C 180,E1 -18808.37,E2 -18808.37} C_VEL
LIN {X 0,Y 247.025,Z 471.855,A -85,B 0,C 180,E1 -18810,E2 -18810} C_VEL
LIN {X 0,Y 247.012,Z 471.23,A -85,B 0,C 180,E1 -18811.63,E2 -18811.63} C_VEL
LIN {X 0,Y 246.934,Z 470.199,A -85,B 0,C 180,E1 -18813.263,E2 -18813.263} C_VEL
LIN {X 0,Y 246.939,Z 468.611,A -85,B 0,C 180,E1 -18814.985,E2 -18814.985} C_VEL
LIN {X 0,Y 247.134,Z 465.645,A -85,B 0,C 180,E1 -18817.352,E2 -18817.352} C_VEL
LIN {X 0,Y 247.551,Z 461.487,A -85,B 0,C 180,E1 -18819.807,E2 -18819.807} C_VEL
LIN {X 0,Y 248.386,Z 455.09,A -85,B 0,C 180,E1 -18822.667,E2 -18822.667} C_VEL
LIN {X 0,Y 249.694,Z 448.121,A -85,B 0,C 180,E1 -18825.091,E2 -18825.091} C_VEL
LIN {X 0,Y 251.013,Z 440.98,A -85,B 0,C 180,E1 -18827.096,E2 -18827.096} C_VEL
LIN {X 0,Y 252.342,Z 432.973,A -85,B 0,C 180,E1 -18828.957,E2 -18828.957} C_VEL
LIN {X 0,Y 254.107,Z 422.818,A -85,B 0,C 180,E1 -18830.86,E2 -18830.86} C_VEL
LIN {X 0,Y 255.776,Z 412.485,A -85,B 0,C 180,E1 -18832.41,E2 -18832.41} C_VEL
LIN {X 0,Y 257.456,Z 401.221,A -85,B 0,C 180,E1 -18833.743,E2 -18833.743} C_VEL
LIN {X 0,Y 259.081,Z 388.612,A -85,B 0,C 180,E1 -18834.863,E2 -18834.863} C_VEL
LIN {X 0,Y 260.203,Z 376.137,A -85,B 0,C 180,E1 -18835.657,E2 -18835.657} C_VEL
LIN {X 0,Y 261.017,Z 362.329,A -85,B 0,C 180,E1 -18836.215,E2 -18836.215} C_VEL
LIN {X 0,Y 262.714,Z 309.55,A -85,B 0,C 180,E1 -18837.735,E2 -18837.735} C_VEL
LIN {X 0,Y 258.12,Z 275.532,A -85,B 0,C 180,E1 -18839.28,E2 -18839.28} C_VEL
LIN {X 0,Y 253.62,Z 262.713,A -85,B 0,C 180,E1 -18840.17,E2 -18840.17} C_VEL
LIN {X 0,Y 252.579,Z 259.858,A -85,B 0,C 180,E1 -18840.381,E2 -18840.381} C_VEL
LIN {X 0,Y 250.491,Z 249.807,A -85,B 0,C 180,E1 -18844.134,E2 -18844.134} C_VEL
LIN {X 0,Y 249.082,Z 243.456,A -85,B 0,C 180,E1 -18846.71,E2 -18846.71} C_VEL
LIN {X 0,Y 248.984,Z 243.474,A -85,B 0,C 180,E1 -18850.481,E2 -18850.481} C_VEL
LIN {X 0,Y 248.958,Z 243.476,A -85,B 0,C 180,E1 -18855.101,E2 -18855.101} C_VEL
LIN {X 0,Y 248.986,Z 243.472,A -85,B 0,C 180,E1 -18859.649,E2 -18859.649} C_VEL
LIN {X 0,Y 249.024,Z 243.466,A -85,B 0,C 180,E1 -18863.645,E2 -18863.645} C_VEL
LIN {X 0,Y 249.008,Z 243.469,A -85,B 0,C 180,E1 -18867.562,E2 -18867.562} C_VEL
LIN {X 0,Y 249.043,Z 243.464,A -85,B 0,C 180,E1 -18871.323,E2 -18871.323} C_VEL
LIN {X 0,Y 249.063,Z 243.458,A -85,B 0,C 180,E1 -18874.951,E2 -18874.951} C_VEL
LIN {X 0,Y 249.057,Z 243.456,A -85,B 0,C 180,E1 -18878.62,E2 -18878.62} C_VEL
LIN {X 0,Y 249.162,Z 243.433,A -85,B 0,C 180,E1 -18883.608,E2 -18883.608} C_VEL
LIN {X 0,Y 249.186,Z 243.442,A -85,B 0,C 180,E1 -18886.951,E2 -18886.951} C_VEL
LIN {X 0,Y 249.372,Z 243.418,A -85,B 0,C 180,E1 -18890.53,E2 -18890.53} C_VEL
LIN {X 0,Y 249.416,Z 243.404,A -85,B 0,C 180,E1 -18893.52,E2 -18893.52} C_VEL
LIN {X 0,Y 249.642,Z 243.369,A -85,B 0,C 180,E1 -18898.378,E2 -18898.378} C_VEL
LIN {X 0,Y 249.649,Z 243.383,A -85,B 0,C 180,E1 -18901.604,E2 -18901.604} C_VEL
LIN {X 0,Y 249.408,Z 243.414,A -85,B 0,C 180,E1 -18906.537,E2 -18906.537} C_VEL
LIN {X 0,Y 249.33,Z 243.421,A -85,B 0,C 180,E1 -18909.727,E2 -18909.727} C_VEL
LIN {X 0,Y 249.164,Z 243.446,A -85,B 0,C 180,E1 -18914.695,E2 -18914.695} C_VEL
LIN {X 0,Y 249.101,Z 243.446,A -85,B 0,C 180,E1 -18918.069,E2 -18918.069} C_VEL
LIN {X 0,Y 249.063,Z 243.461,A -85,B 0,C 180,E1 -18921.509,E2 -18921.509} C_VEL
LIN {X 0,Y 249.087,Z 243.454,A -85,B 0,C 180,E1 -18925.464,E2 -18925.464} C_VEL
LIN {X 0,Y 249.026,Z 243.449,A -85,B 0,C 180,E1 -18928.972,E2 -18928.972} C_VEL
LIN {X 0,Y 248.997,Z 243.443,A -85,B 0,C 180,E1 -18932.418,E2 -18932.418} C_VEL
LIN {X 0,Y 248.993,Z 243.462,A -85,B 0,C 180,E1 -18936.338,E2 -18936.338} C_VEL
LIN {X 0,Y 248.956,Z 243.472,A -85,B 0,C 180,E1 -18940.473,E2 -18940.473} C_VEL
LIN {X 0,Y 248.972,Z 243.468,A -85,B 0,C 180,E1 -18942.785,E2 -18942.785} C_VEL
LIN {X 0,Y 248.977,Z 243.473,A -85,B 0,C 180,E1 -18947.356,E2 -18947.356} C_VEL
LIN {X 0,Y 249,Z 243.466,A -85,B 0,C 180,E1 -18952.194,E2 -18952.194} C_VEL
LIN {X 0,Y 248.998,Z 243.466,A -85,B 0,C 180,E1 -18955.633,E2 -18955.633} C_VEL
LIN {X 0,Y 249.004,Z 243.471,A -85,B 0,C 180,E1 -18959.467,E2 -18959.467} C_VEL
LIN {X 0,Y 249.028,Z 243.466,A -85,B 0,C 180,E1 -18963.158,E2 -18963.158} C_VEL
LIN {X 0,Y 249.064,Z 243.463,A -85,B 0,C 180,E1 -18966.732,E2 -18966.732} C_VEL
LIN {X 0,Y 249.096,Z 243.458,A -85,B 0,C 180,E1 -18970.211,E2 -18970.211} C_VEL
LIN {X 0,Y 249.191,Z 243.447,A -85,B 0,C 180,E1 -18973.619,E2 -18973.619} C_VEL
LIN {X 0,Y 249.198,Z 243.444,A -85,B 0,C 180,E1 -18978.614,E2 -18978.614} C_VEL
LIN {X 0,Y 249.428,Z 243.413,A -85,B 0,C 180,E1 -18981.901,E2 -18981.901} C_VEL
LIN {X 0,Y 249.411,Z 243.416,A -85,B 0,C 180,E1 -18986.769,E2 -18986.769} C_VEL
LIN {X 0,Y 249.68,Z 243.382,A -85,B 0,C 180,E1 -18990,E2 -18990} C_VEL
LIN {X 0,Y 249.549,Z 243.398,A -85,B 0,C 180,E1 -18992.371,E2 -18992.371} C_VEL
LIN {X 0,Y 250.625,Z 246.421,A -85,B 0,C 180,E1 -18992.607,E2 -18992.607} C_VEL
LIN {X 0,Y 258.87,Z 266.656,A -85,B 0,C 180,E1 -18994.145,E2 -18994.145} C_VEL
LIN {X 0,Y 263.653,Z 280.476,A -85,B 0,C 180,E1 -18995.063,E2 -18995.063} C_VEL
LIN {X 0,Y 261.042,Z 350.999,A -85,B 0,C 180,E1 -18997.114,E2 -18997.114} C_VEL
LIN {X 0,Y 260.125,Z 363.617,A -85,B 0,C 180,E1 -18997.763,E2 -18997.763} C_VEL
LIN {X 0,Y 258.978,Z 376.835,A -85,B 0,C 180,E1 -18998.78,E2 -18998.78} C_VEL
LIN {X 0,Y 257.546,Z 388.446,A -85,B 0,C 180,E1 -18999.991,E2 -18999.991} C_VEL
LIN {X 0,Y 255.975,Z 399.556,A -85,B 0,C 180,E1 -19001.481,E2 -19001.481} C_VEL
LIN {X 0,Y 254.144,Z 410.542,A -85,B 0,C 180,E1 -19003.339,E2 -19003.339} C_VEL
LIN {X 0,Y 252.382,Z 419.925,A -85,B 0,C 180,E1 -19005.339,E2 -19005.339} C_VEL
LIN {X 0,Y 250.804,Z 428.863,A -85,B 0,C 180,E1 -19007.725,E2 -19007.725} C_VEL
LIN {X 0,Y 249.481,Z 436.042,A -85,B 0,C 180,E1 -19010.136,E2 -19010.136} C_VEL
LIN {X 0,Y 248.514,Z 441.512,A -85,B 0,C 180,E1 -19012.443,E2 -19012.443} C_VEL
LIN {X 0,Y 247.735,Z 446.53,A -85,B 0,C 180,E1 -19015.184,E2 -19015.184} C_VEL
LIN {X 0,Y 247.392,Z 449.162,A -85,B 0,C 180,E1 -19017.034,E2 -19017.034} C_VEL
LIN {X 0,Y 246.984,Z 451.21,A -85,B 0,C 180,E1 -19018.929,E2 -19018.929} C_VEL
LIN {X 0,Y 246.694,Z 452.994,A -85,B 0,C 180,E1 -19021.301,E2 -19021.301} C_VEL
LIN {X 0,Y 246.656,Z 454.001,A -85,B 0,C 180,E1 -19024.301,E2 -19024.301} C_VEL
LIN {X 0,Y 246.98,Z 453.707,A -85,B 0,C 180,E1 -19027.198,E2 -19027.198} C_VEL
LIN {X 0,Y 247.63,Z 452.227,A -85,B 0,C 180,E1 -19029.997,E2 -19029.997} C_VEL
LIN {X 0,Y 248.557,Z 449.586,A -85,B 0,C 180,E1 -19032.733,E2 -19032.733} C_VEL
LIN {X 0,Y 249.813,Z 445.902,A -85,B 0,C 180,E1 -19035.322,E2 -19035.322} C_VEL
LIN {X 0,Y 251.322,Z 441.047,A -85,B 0,C 180,E1 -19037.86,E2 -19037.86} C_VEL
LIN {X 0,Y 253.293,Z 434.832,A -85,B 0,C 180,E1 -19040.359,E2 -19040.359} C_VEL
LIN {X 0,Y 255.747,Z 426.945,A -85,B 0,C 180,E1 -19042.836,E2 -19042.836} C_VEL
LIN {X 0,Y 257.995,Z 419.042,A -85,B 0,C 180,E1 -19044.806,E2 -19044.806} C_VEL
LIN {X 0,Y 260.496,Z 409.313,A -85,B 0,C 180,E1 -19046.755,E2 -19046.755} C_VEL
LIN {X 0,Y 262.997,Z 398.405,A -85,B 0,C 180,E1 -19048.493,E2 -19048.493} C_VEL
LIN {X 0,Y 265.157,Z 387.204,A -85,B 0,C 180,E1 -19049.889,E2 -19049.889} C_VEL
LIN {X 0,Y 267.078,Z 375.329,A -85,B 0,C 180,E1 -19051.015,E2 -19051.015} C_VEL
LIN {X 0,Y 268.619,Z 362.478,A -85,B 0,C 180,E1 -19051.916,E2 -19051.916} C_VEL
LIN {X 0,Y 269.698,Z 349.355,A -85,B 0,C 180,E1 -19052.511,E2 -19052.511} C_VEL
LIN {X 0,Y 272.617,Z 287.942,A -85,B 0,C 180,E1 -19054.271,E2 -19054.271} C_VEL
LIN {X 0,Y 266.733,Z 274.53,A -85,B 0,C 180,E1 -19055.753,E2 -19055.753} C_VEL
LIN {X 0,Y 259.809,Z 261.401,A -85,B 0,C 180,E1 -19057.548,E2 -19057.548} C_VEL
LIN {X 0,Y 254.254,Z 252.461,A -85,B 0,C 180,E1 -19059.057,E2 -19059.057} C_VEL
LIN {X 0,Y 250.969,Z 247.39,A -85,B 0,C 180,E1 -19060.002,E2 -19060.002} C_VEL
LIN {X 0,Y 249.352,Z 244.548,A -85,B 0,C 180,E1 -19060.564,E2 -19060.564} C_VEL
LIN {X 0,Y 249.121,Z 243.457,A -85,B 0,C 180,E1 -19061.187,E2 -19061.187} C_VEL
LIN {X 0,Y 249.224,Z 243.443,A -85,B 0,C 180,E1 -19063.631,E2 -19063.631} C_VEL
